LIN {X 0,Y 309.952,Z 757.671,A -85,B 0,C 180,E1 16400.5,E2 16400.5} C_VEL
LIN {X 0,Y 315.496,Z 768.364,A -85,B 0,C 180,E1 16405.207,E2 16405.207} C_VEL
LIN {X 0,Y 323.585,Z 785.947,A -85,B 0,C 180,E1 16410.491,E2 16410.491} C_VEL
LIN {X 0,Y 330.454,Z 808.188,A -85,B 0,C 180,E1 16415.117,E2 16415.117} C_VEL
LIN {X 0,Y 332.318,Z 818.689,A -85,B 0,C 180,E1 16416.877,E2 16416.877} C_VEL
LIN {X 0,Y 321.073,Z 855.454,A -85,B 0,C 180,E1 16419.899,E2 16419.899} C_VEL
LIN {X 0,Y 307.71,Z 890.699,A -85,B 0,C 180,E1 16424.174,E2 16424.174} C_VEL
LIN {X 0,Y 294.928,Z 920.705,A -85,B 0,C 180,E1 16429.49,E2 16429.49} C_VEL
LIN {X 0,Y 283.712,Z 946.43,A -85,B 0,C 180,E1 16435.988,E2 16435.988} C_VEL
LIN {X 0,Y 275.518,Z 966.441,A -85,B 0,C 180,E1 16443.137,E2 16443.137} C_VEL
LIN {X 0,Y 270.884,Z 980.87,A -85,B 0,C 180,E1 16450.473,E2 16450.473} C_VEL
LIN {X 0,Y 268.893,Z 991.255,A -85,B 0,C 180,E1 16458.671,E2 16458.671} C_VEL
LIN {X 0,Y 268.674,Z 996.154,A -85,B 0,C 180,E1 16466.78,E2 16466.78} C_VEL
LIN {X 0,Y 269.019,Z 996.603,A -85,B 0,C 180,E1 16470,E2 16470} C_VEL
LIN {X 0,Y 268.663,Z 993.875,A -85,B 0,C 180,E1 16478.072,E2 16478.072} C_VEL
LIN {X 0,Y 269.779,Z 985.621,A -85,B 0,C 180,E1 16486.241,E2 16486.241} C_VEL
LIN {X 0,Y 273.628,Z 971.419,A -85,B 0,C 180,E1 16494.444,E2 16494.444} C_VEL
LIN {X 0,Y 280.981,Z 951.52,A -85,B 0,C 180,E1 16502.08,E2 16502.08} C_VEL
LIN {X 0,Y 291.2,Z 926.496,A -85,B 0,C 180,E1 16508.747,E2 16508.747} C_VEL
LIN {X 0,Y 302.201,Z 899.005,A -85,B 0,C 180,E1 16513.938,E2 16513.938} C_VEL
LIN {X 0,Y 313.934,Z 866.938,A -85,B 0,C 180,E1 16518.208,E2 16518.208} C_VEL
LIN {X 0,Y 324.235,Z 833.113,A -85,B 0,C 180,E1 16521.361,E2 16521.361} C_VEL
LIN {X 0,Y 328.214,Z 816.116,A -85,B 0,C 180,E1 16522.625,E2 16522.625} C_VEL
LIN {X 0,Y 317.617,Z 786.468,A -85,B 0,C 180,E1 16527.572,E2 16527.572} C_VEL
LIN {X 0,Y 309.539,Z 769.18,A -85,B 0,C 180,E1 16530.843,E2 16530.843} C_VEL
LIN {X 0,Y 305.434,Z 765.763,A -85,B 0,C 180,E1 16532.16,E2 16532.16} C_VEL
LIN {X 0,Y 298.724,Z 762.182,A -85,B 0,C 180,E1 16534.27,E2 16534.27} C_VEL
LIN {X 0,Y 298.214,Z 761.313,A -85,B 0,C 180,E1 16534.479,E2 16534.479} C_VEL
LIN {X 0,Y 284.887,Z 739.622,A -85,B 0,C 180,E1 16540.243,E2 16540.243} C_VEL
LIN {X 0,Y 273.531,Z 723.276,A -85,B 0,C 180,E1 16545.909,E2 16545.909} C_VEL
LIN {X 0,Y 268.525,Z 716.432,A -85,B 0,C 180,E1 16548.856,E2 16548.856} C_VEL
LIN {X 0,Y 265.071,Z 710.925,A -85,B 0,C 180,E1 16551.193,E2 16551.193} C_VEL
LIN {X 0,Y 260.012,Z 704.969,A -85,B 0,C 180,E1 16554.98,E2 16554.98} C_VEL
LIN {X 0,Y 259.721,Z 702.53,A -85,B 0,C 180,E1 16555.809,E2 16555.809} C_VEL
LIN {X 0,Y 260.153,Z 702.53,A -85,B 0,C 180,E1 16559.973,E2 16559.973} C_VEL
LIN {X 0,Y 259.354,Z 702.53,A -85,B 0,C 180,E1 16568.46,E2 16568.46} C_VEL
LIN {X 0,Y 258.71,Z 702.53,A -85,B 0,C 180,E1 16576.924,E2 16576.924} C_VEL
LIN {X 0,Y 258.198,Z 702.53,A -85,B 0,C 180,E1 16584.113,E2 16584.113} C_VEL
LIN {X 0,Y 257.794,Z 702.53,A -85,B 0,C 180,E1 16591.751,E2 16591.751} C_VEL
LIN {X 0,Y 257.771,Z 703.057,A -85,B 0,C 180,E1 16597.239,E2 16597.239} C_VEL
LIN {X 0,Y 259.94,Z 708.124,A -85,B 0,C 180,E1 16599.361,E2 16599.361} C_VEL
LIN {X 0,Y 263.477,Z 711.105,A -85,B 0,C 180,E1 16601.928,E2 16601.928} C_VEL
LIN {X 0,Y 267.434,Z 716.658,A -85,B 0,C 180,E1 16604.625,E2 16604.625} C_VEL
LIN {X 0,Y 278.791,Z 731.981,A -85,B 0,C 180,E1 16611.013,E2 16611.013} C_VEL
LIN {X 0,Y 290.731,Z 751.396,A -85,B 0,C 180,E1 16617.012,E2 16617.012} C_VEL
LIN {X 0,Y 301.764,Z 773.502,A -85,B 0,C 180,E1 16622.492,E2 16622.492} C_VEL
LIN {X 0,Y 310.582,Z 798.842,A -85,B 0,C 180,E1 16627.717,E2 16627.717} C_VEL
LIN {X 0,Y 313.35,Z 812.889,A -85,B 0,C 180,E1 16630.3,E2 16630.3} C_VEL
LIN {X 0,Y 302.475,Z 846.573,A -85,B 0,C 180,E1 16634.075,E2 16634.075} C_VEL
LIN {X 0,Y 291.256,Z 875.538,A -85,B 0,C 180,E1 16638.797,E2 16638.797} C_VEL
LIN {X 0,Y 280.621,Z 900.044,A -85,B 0,C 180,E1 16644.533,E2 16644.533} C_VEL
LIN {X 0,Y 271.528,Z 920.415,A -85,B 0,C 180,E1 16651.468,E2 16651.468} C_VEL
LIN {X 0,Y 265.354,Z 935.057,A -85,B 0,C 180,E1 16658.959,E2 16658.959} C_VEL
LIN {X 0,Y 262.16,Z 944.332,A -85,B 0,C 180,E1 16666.727,E2 16666.727} C_VEL
LIN {X 0,Y 260.433,Z 948.523,A -85,B 0,C 180,E1 16673.929,E2 16673.929} C_VEL
LIN {X 0,Y 260.646,Z 948.698,A -85,B 0,C 180,E1 16681.404,E2 16681.404} C_VEL
LIN {X 0,Y 263.067,Z 944.4,A -85,B 0,C 180,E1 16689.124,E2 16689.124} C_VEL
LIN {X 0,Y 267.8,Z 934.327,A -85,B 0,C 180,E1 16697.501,E2 16697.501} C_VEL
LIN {X 0,Y 275.753,Z 918.84,A -85,B 0,C 180,E1 16705.171,E2 16705.171} C_VEL
LIN {X 0,Y 286.314,Z 898.705,A -85,B 0,C 180,E1 16711.718,E2 16711.718} C_VEL
LIN {X 0,Y 298.719,Z 873.349,A -85,B 0,C 180,E1 16717.371,E2 16717.371} C_VEL
LIN {X 0,Y 311.444,Z 844.042,A -85,B 0,C 180,E1 16721.852,E2 16721.852} C_VEL
LIN {X 0,Y 320.875,Z 817.036,A -85,B 0,C 180,E1 16724.861,E2 16724.861} C_VEL
LIN {X 0,Y 317.416,Z 795.177,A -85,B 0,C 180,E1 16729.755,E2 16729.755} C_VEL
LIN {X 0,Y 312.367,Z 777.587,A -85,B 0,C 180,E1 16734.827,E2 16734.827} C_VEL
LIN {X 0,Y 307.316,Z 764.973,A -85,B 0,C 180,E1 16740.239,E2 16740.239} C_VEL
LIN {X 0,Y 305.699,Z 761.257,A -85,B 0,C 180,E1 16742.579,E2 16742.579} C_VEL
LIN {X 0,Y 304.113,Z 756.55,A -85,B 0,C 180,E1 16746.2,E2 16746.2} C_VEL
LIN {X 0,Y 304.093,Z 757.322,A -85,B 0,C 180,E1 16754.463,E2 16754.463} C_VEL
LIN {X 0,Y 307.631,Z 765.127,A -85,B 0,C 180,E1 16760.204,E2 16760.204} C_VEL
LIN {X 0,Y 312.812,Z 776.006,A -85,B 0,C 180,E1 16765.025,E2 16765.025} C_VEL
LIN {X 0,Y 319.966,Z 793.22,A -85,B 0,C 180,E1 16770.23,E2 16770.23} C_VEL
LIN {X 0,Y 325.982,Z 815.534,A -85,B 0,C 180,E1 16774.947,E2 16774.947} C_VEL
LIN {X 0,Y 326.56,Z 822.504,A -85,B 0,C 180,E1 16776.018,E2 16776.018} C_VEL
LIN {X 0,Y 314.643,Z 858.935,A -85,B 0,C 180,E1 16779.172,E2 16779.172} C_VEL
LIN {X 0,Y 301.149,Z 892.374,A -85,B 0,C 180,E1 16783.399,E2 16783.399} C_VEL
LIN {X 0,Y 287.801,Z 922.182,A -85,B 0,C 180,E1 16788.882,E2 16788.882} C_VEL
LIN {X 0,Y 276.655,Z 946.385,A -85,B 0,C 180,E1 16795.212,E2 16795.212} C_VEL
LIN {X 0,Y 267.479,Z 967.633,A -85,B 0,C 180,E1 16803.17,E2 16803.17} C_VEL
LIN {X 0,Y 262.701,Z 981.909,A -85,B 0,C 180,E1 16811.046,E2 16811.046} C_VEL
LIN {X 0,Y 261.036,Z 990.52,A -85,B 0,C 180,E1 16818.282,E2 16818.282} C_VEL
LIN {X 0,Y 260.73,Z 994.111,A -85,B 0,C 180,E1 16823.352,E2 16823.352} C_VEL
LIN {X 0,Y 261.163,Z 995.89,A -85,B 0,C 180,E1 16830,E2 16830} C_VEL
LIN {X 0,Y 260.794,Z 993.127,A -85,B 0,C 180,E1 16838.317,E2 16838.317} C_VEL
LIN {X 0,Y 262.019,Z 984.826,A -85,B 0,C 180,E1 16846.735,E2 16846.735} C_VEL
LIN {X 0,Y 266.059,Z 970.858,A -85,B 0,C 180,E1 16855.021,E2 16855.021} C_VEL
LIN {X 0,Y 273.951,Z 950.669,A -85,B 0,C 180,E1 16862.953,E2 16862.953} C_VEL
LIN {X 0,Y 284.345,Z 926.389,A -85,B 0,C 180,E1 16869.556,E2 16869.556} C_VEL
LIN {X 0,Y 296.508,Z 897.188,A -85,B 0,C 180,E1 16875.123,E2 16875.123} C_VEL
LIN {X 0,Y 308.405,Z 865.604,A -85,B 0,C 180,E1 16879.324,E2 16879.324} C_VEL
LIN {X 0,Y 319.029,Z 831.642,A -85,B 0,C 180,E1 16882.465,E2 16882.465} C_VEL
LIN {X 0,Y 322.022,Z 818.898,A -85,B 0,C 180,E1 16883.439,E2 16883.439} C_VEL
LIN {X 0,Y 312.462,Z 791.073,A -85,B 0,C 180,E1 16888.3,E2 16888.3} C_VEL
LIN {X 0,Y 299.497,Z 763.712,A -85,B 0,C 180,E1 16893.922,E2 16893.922} C_VEL
LIN {X 0,Y 298.214,Z 761.313,A -85,B 0,C 180,E1 16894.479,E2 16894.479} C_VEL
LIN {X 0,Y 292.885,Z 755.46,A -85,B 0,C 180,E1 16896.496,E2 16896.496} C_VEL
LIN {X 0,Y 283.364,Z 748.358,A -85,B 0,C 180,E1 16900.231,E2 16900.231} C_VEL
LIN {X 0,Y 271.288,Z 730.388,A -85,B 0,C 180,E1 16906.474,E2 16906.474} C_VEL
LIN {X 0,Y 265.81,Z 723.086,A -85,B 0,C 180,E1 16909.8,E2 16909.8} C_VEL
LIN {X 0,Y 261.859,Z 717.005,A -85,B 0,C 180,E1 16912.634,E2 16912.634} C_VEL
LIN {X 0,Y 257.895,Z 711.36,A -85,B 0,C 180,E1 16915.885,E2 16915.885} C_VEL
LIN {X 0,Y 255.967,Z 709.404,A -85,B 0,C 180,E1 16917.586,E2 16917.586} C_VEL
LIN {X 0,Y 252.121,Z 703.78,A -85,B 0,C 180,E1 16921.901,E2 16921.901} C_VEL
LIN {X 0,Y 252.032,Z 702.53,A -85,B 0,C 180,E1 16922.546,E2 16922.546} C_VEL
LIN {X 0,Y 251.304,Z 702.53,A -85,B 0,C 180,E1 16930.348,E2 16930.348} C_VEL
LIN {X 0,Y 250.706,Z 702.53,A -85,B 0,C 180,E1 16937.482,E2 16937.482} C_VEL
LIN {X 0,Y 250.123,Z 702.53,A -85,B 0,C 180,E1 16945.182,E2 16945.182} C_VEL
LIN {X 0,Y 249.917,Z 703.282,A -85,B 0,C 180,E1 16949.517,E2 16949.517} C_VEL
LIN {X 0,Y 252.514,Z 708.484,A -85,B 0,C 180,E1 16953.302,E2 16953.302} C_VEL
LIN {X 0,Y 255.955,Z 711.064,A -85,B 0,C 180,E1 16956.691,E2 16956.691} C_VEL
LIN {X 0,Y 259.601,Z 716.781,A -85,B 0,C 180,E1 16959.968,E2 16959.968} C_VEL
LIN {X 0,Y 261.694,Z 719.033,A -85,B 0,C 180,E1 16961.535,E2 16961.535} C_VEL
LIN {X 0,Y 267.398,Z 727.187,A -85,B 0,C 180,E1 16965.485,E2 16965.485} C_VEL
LIN {X 0,Y 276.033,Z 739.146,A -85,B 0,C 180,E1 16970.543,E2 16970.543} C_VEL
LIN {X 0,Y 287.79,Z 759.139,A -85,B 0,C 180,E1 16976.872,E2 16976.872} C_VEL
LIN {X 0,Y 297.989,Z 781.572,A -85,B 0,C 180,E1 16982.479,E2 16982.479} C_VEL
LIN {X 0,Y 305.562,Z 805.841,A -85,B 0,C 180,E1 16987.618,E2 16987.618} C_VEL
LIN {X 0,Y 307.052,Z 816.176,A -85,B 0,C 180,E1 16989.514,E2 16989.514} C_VEL
LIN {X 0,Y 295.398,Z 850.222,A -85,B 0,C 180,E1 16993.492,E2 16993.492} C_VEL
LIN {X 0,Y 283.523,Z 879.262,A -85,B 0,C 180,E1 16998.487,E2 16998.487} C_VEL
LIN {X 0,Y 272.351,Z 904.007,A -85,B 0,C 180,E1 17004.666,E2 17004.666} C_VEL
LIN {X 0,Y 263.492,Z 922.835,A -85,B 0,C 180,E1 17011.512,E2 17011.512} C_VEL
LIN {X 0,Y 257.221,Z 937.08,A -85,B 0,C 180,E1 17019.392,E2 17019.392} C_VEL
LIN {X 0,Y 254.111,Z 945.653,A -85,B 0,C 180,E1 17027.273,E2 17027.273} C_VEL
LIN {X 0,Y 252.449,Z 949.511,A -85,B 0,C 180,E1 17034.736,E2 17034.736} C_VEL
LIN {X 0,Y 253.221,Z 948.827,A -85,B 0,C 180,E1 17043.527,E2 17043.527} C_VEL
LIN {X 0,Y 255.721,Z 944.406,A -85,B 0,C 180,E1 17050.476,E2 17050.476} C_VEL
LIN {X 0,Y 260.915,Z 934.25,A -85,B 0,C 180,E1 17058.753,E2 17058.753} C_VEL
LIN {X 0,Y 269.311,Z 919,A -85,B 0,C 180,E1 17066.295,E2 17066.295} C_VEL
LIN {X 0,Y 280.66,Z 898.461,A -85,B 0,C 180,E1 17073.015,E2 17073.015} C_VEL
LIN {X 0,Y 293.25,Z 873.912,A -85,B 0,C 180,E1 17078.513,E2 17078.513} C_VEL
LIN {X 0,Y 306.964,Z 843.551,A -85,B 0,C 180,E1 17083.153,E2 17083.153} C_VEL
LIN {X 0,Y 315.393,Z 819.76,A -85,B 0,C 180,E1 17085.892,E2 17085.892} C_VEL
LIN {X 0,Y 312.425,Z 798.271,A -85,B 0,C 180,E1 17090.993,E2 17090.993} C_VEL
LIN {X 0,Y 308.013,Z 781.769,A -85,B 0,C 180,E1 17096.224,E2 17096.224} C_VEL
LIN {X 0,Y 303.922,Z 769.5,A -85,B 0,C 180,E1 17101.908,E2 17101.908} C_VEL
LIN {X 0,Y 301.889,Z 764.119,A -85,B 0,C 180,E1 17106.733,E2 17106.733} C_VEL
LIN {X 0,Y 302.054,Z 764.998,A -85,B 0,C 180,E1 17114.258,E2 17114.258} C_VEL
LIN {X 0,Y 305.197,Z 772.567,A -85,B 0,C 180,E1 17119.964,E2 17119.964} C_VEL
LIN {X 0,Y 310.416,Z 784.431,A -85,B 0,C 180,E1 17125.192,E2 17125.192} C_VEL
LIN {X 0,Y 316.779,Z 802.18,A -85,B 0,C 180,E1 17130.426,E2 17130.426} C_VEL
LIN {X 0,Y 321.468,Z 823.556,A -85,B 0,C 180,E1 17134.913,E2 17134.913} C_VEL
LIN {X 0,Y 308.737,Z 860.849,A -85,B 0,C 180,E1 17138.245,E2 17138.245} C_VEL
LIN {X 0,Y 295.1,Z 893.08,A -85,B 0,C 180,E1 17142.425,E2 17142.425} C_VEL
LIN {X 0,Y 281.395,Z 922.208,A -85,B 0,C 180,E1 17147.907,E2 17147.907} C_VEL
LIN {X 0,Y 269.669,Z 946.291,A -85,B 0,C 180,E1 17154.376,E2 17154.376} C_VEL
LIN {X 0,Y 260.182,Z 966.977,A -85,B 0,C 180,E1 17162.355,E2 17162.355} C_VEL
LIN {X 0,Y 254.987,Z 981.316,A -85,B 0,C 180,E1 17170.512,E2 17170.512} C_VEL
LIN {X 0,Y 253.174,Z 989.86,A -85,B 0,C 180,E1 17177.958,E2 17177.958} C_VEL
LIN {X 0,Y 252.865,Z 993.419,A -85,B 0,C 180,E1 17183.145,E2 17183.145} C_VEL
LIN {X 0,Y 253.293,Z 995.176,A -85,B 0,C 180,E1 17190,E2 17190} C_VEL
LIN {X 0,Y 252.915,Z 992.371,A -85,B 0,C 180,E1 17198.578,E2 17198.578} C_VEL
LIN {X 0,Y 254.261,Z 984.005,A -85,B 0,C 180,E1 17207.262,E2 17207.262} C_VEL
LIN {X 0,Y 258.795,Z 969.492,A -85,B 0,C 180,E1 17216.009,E2 17216.009} C_VEL
LIN {X 0,Y 267.032,Z 949.646,A -85,B 0,C 180,E1 17223.92,E2 17223.92} C_VEL
LIN {X 0,Y 278.05,Z 925.23,A -85,B 0,C 180,E1 17230.636,E2 17230.636} C_VEL
LIN {X 0,Y 290.412,Z 896.619,A -85,B 0,C 180,E1 17236.149,E2 17236.149} C_VEL
LIN {X 0,Y 302.589,Z 865.36,A -85,B 0,C 180,E1 17240.342,E2 17240.342} C_VEL
LIN {X 0,Y 314.007,Z 829.906,A -85,B 0,C 180,E1 17243.622,E2 17243.622} C_VEL
LIN {X 0,Y 315.829,Z 821.525,A -85,B 0,C 180,E1 17244.316,E2 17244.316} C_VEL
LIN {X 0,Y 306.732,Z 794.337,A -85,B 0,C 180,E1 17249.29,E2 17249.29} C_VEL
LIN {X 0,Y 294.241,Z 767.159,A -85,B 0,C 180,E1 17255.152,E2 17255.152} C_VEL
LIN {X 0,Y 283.364,Z 748.358,A -85,B 0,C 180,E1 17260.231,E2 17260.231} C_VEL
LIN {X 0,Y 276.578,Z 742.524,A -85,B 0,C 180,E1 17263.301,E2 17263.301} C_VEL
LIN {X 0,Y 269.757,Z 738.248,A -85,B 0,C 180,E1 17266.613,E2 17266.613} C_VEL
LIN {X 0,Y 259.79,Z 724.228,A -85,B 0,C 180,E1 17273.303,E2 17273.303} C_VEL
LIN {X 0,Y 255.908,Z 718.162,A -85,B 0,C 180,E1 17276.669,E2 17276.669} C_VEL
LIN {X 0,Y 250.725,Z 711.765,A -85,B 0,C 180,E1 17282.235,E2 17282.235} C_VEL
LIN {X 0,Y 249.92,Z 710.151,A -85,B 0,C 180,E1 17283.433,E2 17283.433} C_VEL
LIN {X 0,Y 244.951,Z 707.669,A -85,B 0,C 180,E1 17294.233,E2 17294.233} C_VEL
LIN {X 0,Y 248.352,Z 710.423,A -85,B 0,C 180,E1 17308.742,E2 17308.742} C_VEL
LIN {X 0,Y 251.252,Z 716.251,A -85,B 0,C 180,E1 17313.123,E2 17313.123} C_VEL
LIN {X 0,Y 254.28,Z 718.794,A -85,B 0,C 180,E1 17316.226,E2 17316.226} C_VEL
LIN {X 0,Y 258.378,Z 724.622,A -85,B 0,C 180,E1 17319.928,E2 17319.928} C_VEL
LIN {X 0,Y 265.434,Z 734.864,A -85,B 0,C 180,E1 17325.172,E2 17325.172} C_VEL
LIN {X 0,Y 273.871,Z 747.567,A -85,B 0,C 180,E1 17330.502,E2 17330.502} C_VEL
LIN {X 0,Y 283.765,Z 765.176,A -85,B 0,C 180,E1 17336.237,E2 17336.237} C_VEL
LIN {X 0,Y 292.976,Z 786.556,A -85,B 0,C 180,E1 17341.778,E2 17341.778} C_VEL
LIN {X 0,Y 299.743,Z 809.701,A -85,B 0,C 180,E1 17346.885,E2 17346.885} C_VEL
LIN {X 0,Y 300.903,Z 819.016,A -85,B 0,C 180,E1 17348.658,E2 17348.658} C_VEL
LIN {X 0,Y 288.794,Z 852.607,A -85,B 0,C 180,E1 17352.712,E2 17352.712} C_VEL
LIN {X 0,Y 276.601,Z 881.237,A -85,B 0,C 180,E1 17357.796,E2 17357.796} C_VEL
LIN {X 0,Y 264.9,Z 906.018,A -85,B 0,C 180,E1 17364.221,E2 17364.221} C_VEL
LIN {X 0,Y 255.917,Z 924.145,A -85,B 0,C 180,E1 17371.114,E2 17371.114} C_VEL
LIN {X 0,Y 249.212,Z 938.66,A -85,B 0,C 180,E1 17379.586,E2 17379.586} C_VEL
LIN {X 0,Y 246.057,Z 946.935,A -85,B 0,C 180,E1 17387.857,E2 17387.857} C_VEL
LIN {X 0,Y 244.507,Z 950.35,A -85,B 0,C 180,E1 17395.596,E2 17395.596} C_VEL
LIN {X 0,Y 245.381,Z 949.643,A -85,B 0,C 180,E1 17403.606,E2 17403.606} C_VEL
LIN {X 0,Y 248.46,Z 944.323,A -85,B 0,C 180,E1 17411.92,E2 17411.92} C_VEL
LIN {X 0,Y 254.508,Z 933.497,A -85,B 0,C 180,E1 17420.426,E2 17420.426} C_VEL
LIN {X 0,Y 263.868,Z 917.609,A -85,B 0,C 180,E1 17428.111,E2 17428.111} C_VEL
LIN {X 0,Y 276.714,Z 895.521,A -85,B 0,C 180,E1 17435.106,E2 17435.106} C_VEL
LIN {X 0,Y 290.617,Z 869.15,A -85,B 0,C 180,E1 17440.664,E2 17440.664} C_VEL
LIN {X 0,Y 304.031,Z 839.579,A -85,B 0,C 180,E1 17444.915,E2 17444.915} C_VEL
LIN {X 0,Y 310.084,Z 823.602,A -85,B 0,C 180,E1 17446.732,E2 17446.732} C_VEL
LIN {X 0,Y 307.824,Z 802.789,A -85,B 0,C 180,E1 17451.923,E2 17451.923} C_VEL
LIN {X 0,Y 304.146,Z 787.118,A -85,B 0,C 180,E1 17457.18,E2 17457.18} C_VEL
LIN {X 0,Y 300.784,Z 776.165,A -85,B 0,C 180,E1 17462.898,E2 17462.898} C_VEL
LIN {X 0,Y 299.708,Z 771.704,A -85,B 0,C 180,E1 17466.527,E2 17466.527} C_VEL
LIN {X 0,Y 299.751,Z 772.559,A -85,B 0,C 180,E1 17474.071,E2 17474.071} C_VEL
LIN {X 0,Y 302.518,Z 779.708,A -85,B 0,C 180,E1 17479.581,E2 17479.581} C_VEL
LIN {X 0,Y 307.375,Z 792.005,A -85,B 0,C 180,E1 17485.07,E2 17485.07} C_VEL
LIN {X 0,Y 312.916,Z 809.903,A -85,B 0,C 180,E1 17490.307,E2 17490.307} C_VEL
LIN {X 0,Y 315.904,Z 826.108,A -85,B 0,C 180,E1 17493.842,E2 17493.842} C_VEL
LIN {X 0,Y 303.741,Z 860.867,A -85,B 0,C 180,E1 17497.084,E2 17497.084} C_VEL
LIN {X 0,Y 289.793,Z 892.456,A -85,B 0,C 180,E1 17501.198,E2 17501.198} C_VEL
LIN {X 0,Y 275.329,Z 921.716,A -85,B 0,C 180,E1 17506.756,E2 17506.756} C_VEL
LIN {X 0,Y 262.621,Z 946.496,A -85,B 0,C 180,E1 17513.582,E2 17513.582} C_VEL
LIN {X 0,Y 252.957,Z 966.354,A -85,B 0,C 180,E1 17521.494,E2 17521.494} C_VEL
LIN {X 0,Y 246.907,Z 982.098,A -85,B 0,C 180,E1 17530.925,E2 17530.925} C_VEL
LIN {X 0,Y 245.083,Z 991.181,A -85,B 0,C 180,E1 17540.201,E2 17540.201} C_VEL
LIN {X 0,Y 245,Z 994.042,A -85,B 0,C 180,E1 17546.468,E2 17546.468} C_VEL
LIN {X 0,Y 245.435,Z 994.461,A -85,B 0,C 180,E1 17550,E2 17550} C_VEL
LIN {X 0,Y 244.987,Z 992.571,A -85,B 0,C 180,E1 17557.076,E2 17557.076} C_VEL
LIN {X 0,Y 245.63,Z 987.23,A -85,B 0,C 180,E1 17564.225,E2 17564.225} C_VEL
LIN {X 0,Y 248.901,Z 975.286,A -85,B 0,C 180,E1 17573.208,E2 17573.208} C_VEL
LIN {X 0,Y 256.434,Z 956.837,A -85,B 0,C 180,E1 17581.979,E2 17581.979} C_VEL
LIN {X 0,Y 267.09,Z 933.964,A -85,B 0,C 180,E1 17589.322,E2 17589.322} C_VEL
LIN {X 0,Y 279.965,Z 906.038,A -85,B 0,C 180,E1 17595.495,E2 17595.495} C_VEL
LIN {X 0,Y 292.999,Z 875.279,A -85,B 0,C 180,E1 17600.182,E2 17600.182} C_VEL
LIN {X 0,Y 304.946,Z 841.582,A -85,B 0,C 180,E1 17603.747,E2 17603.747} C_VEL
LIN {X 0,Y 309.885,Z 824.82,A -85,B 0,C 180,E1 17605.101,E2 17605.101} C_VEL
LIN {X 0,Y 301.092,Z 797.494,A -85,B 0,C 180,E1 17610.317,E2 17610.317} C_VEL
LIN {X 0,Y 288.674,Z 769.981,A -85,B 0,C 180,E1 17616.592,E2 17616.592} C_VEL
LIN {X 0,Y 275.983,Z 748.133,A -85,B 0,C 180,E1 17623.091,E2 17623.091} C_VEL
LIN {X 0,Y 269.757,Z 738.248,A -85,B 0,C 180,E1 17626.613,E2 17626.613} C_VEL
LIN {X 0,Y 258.21,Z 731.808,A -85,B 0,C 180,E1 17633.643,E2 17633.643} C_VEL
LIN {X 0,Y 253.05,Z 724.683,A -85,B 0,C 180,E1 17638.264,E2 17638.264} C_VEL
LIN {X 0,Y 248.84,Z 717.96,A -85,B 0,C 180,E1 17643.448,E2 17643.448} C_VEL
LIN {X 0,Y 243.879,Z 715.499,A -85,B 0,C 180,E1 17654.297,E2 17654.297} C_VEL
LIN {X 0,Y 246.955,Z 718.182,A -85,B 0,C 180,E1 17668.28,E2 17668.28} C_VEL
LIN {X 0,Y 250.535,Z 724.433,A -85,B 0,C 180,E1 17673.557,E2 17673.557} C_VEL
LIN {X 0,Y 252.651,Z 726.565,A -85,B 0,C 180,E1 17675.835,E2 17675.835} C_VEL
LIN {X 0,Y 258.317,Z 734.997,A -85,B 0,C 180,E1 17681.04,E2 17681.04} C_VEL
LIN {X 0,Y 266.292,Z 746.827,A -85,B 0,C 180,E1 17686.978,E2 17686.978} C_VEL
LIN {X 0,Y 276.421,Z 764.625,A -85,B 0,C 180,E1 17693.581,E2 17693.581} C_VEL
LIN {X 0,Y 285.997,Z 785.88,A -85,B 0,C 180,E1 17699.704,E2 17699.704} C_VEL
LIN {X 0,Y 293.135,Z 809.737,A -85,B 0,C 180,E1 17705.315,E2 17705.315} C_VEL
LIN {X 0,Y 294.696,Z 821.987,A -85,B 0,C 180,E1 17707.799,E2 17707.799} C_VEL
LIN {X 0,Y 282.752,Z 853.793,A -85,B 0,C 180,E1 17711.727,E2 17711.727} C_VEL
LIN {X 0,Y 270.433,Z 881.631,A -85,B 0,C 180,E1 17716.737,E2 17716.737} C_VEL
LIN {X 0,Y 258.102,Z 906.67,A -85,B 0,C 180,E1 17723.324,E2 17723.324} C_VEL
LIN {X 0,Y 248.302,Z 925.503,A -85,B 0,C 180,E1 17730.722,E2 17730.722} C_VEL
LIN {X 0,Y 241.656,Z 939.199,A -85,B 0,C 180,E1 17738.982,E2 17738.982} C_VEL
LIN {X 0,Y 238.602,Z 946.777,A -85,B 0,C 180,E1 17746.382,E2 17746.382} C_VEL
LIN {X 0,Y 236.947,Z 950.212,A -85,B 0,C 180,E1 17752.465,E2 17752.465} C_VEL
LIN {X 0,Y 236.854,Z 951.194,A -85,B 0,C 180,E1 17760.644,E2 17760.644} C_VEL
LIN {X 0,Y 239.432,Z 947.77,A -85,B 0,C 180,E1 17769.069,E2 17769.069} C_VEL
LIN {X 0,Y 244.935,Z 938.247,A -85,B 0,C 180,E1 17778.562,E2 17778.562} C_VEL
LIN {X 0,Y 253.443,Z 924.575,A -85,B 0,C 180,E1 17786.469,E2 17786.469} C_VEL
LIN {X 0,Y 265.227,Z 905.679,A -85,B 0,C 180,E1 17793.589,E2 17793.589} C_VEL
LIN {X 0,Y 279.832,Z 880.572,A -85,B 0,C 180,E1 17799.879,E2 17799.879} C_VEL
LIN {X 0,Y 294.79,Z 850.899,A -85,B 0,C 180,E1 17804.799,E2 17804.799} C_VEL
LIN {X 0,Y 304.568,Z 827.906,A -85,B 0,C 180,E1 17807.525,E2 17807.525} C_VEL
LIN {X 0,Y 303.517,Z 809.682,A -85,B 0,C 180,E1 17812.167,E2 17812.167} C_VEL
LIN {X 0,Y 300.914,Z 794.958,A -85,B 0,C 180,E1 17817.149,E2 17817.149} C_VEL
LIN {X 0,Y 298.117,Z 783.656,A -85,B 0,C 180,E1 17822.924,E2 17822.924} C_VEL
LIN {X 0,Y 297.227,Z 780.292,A -85,B 0,C 180,E1 17825.85,E2 17825.85} C_VEL
LIN {X 0,Y 296.852,Z 779.072,A -85,B 0,C 180,E1 17831.753,E2 17831.753} C_VEL
LIN {X 0,Y 297.389,Z 781.231,A -85,B 0,C 180,E1 17834.718,E2 17834.718} C_VEL
LIN {X 0,Y 299.554,Z 786.632,A -85,B 0,C 180,E1 17839.133,E2 17839.133} C_VEL
LIN {X 0,Y 303.771,Z 798.613,A -85,B 0,C 180,E1 17844.609,E2 17844.609} C_VEL
LIN {X 0,Y 308.305,Z 815.126,A -85,B 0,C 180,E1 17849.622,E2 17849.622} C_VEL
LIN {X 0,Y 310.551,Z 830.396,A -85,B 0,C 180,E1 17853.046,E2 17853.046} C_VEL
LIN {X 0,Y 296.032,Z 867.528,A -85,B 0,C 180,E1 17856.595,E2 17856.595} C_VEL
LIN {X 0,Y 280.858,Z 899.613,A -85,B 0,C 180,E1 17861.217,E2 17861.217} C_VEL
LIN {X 0,Y 266.023,Z 927.583,A -85,B 0,C 180,E1 17867.101,E2 17867.101} C_VEL
LIN {X 0,Y 253.057,Z 951.454,A -85,B 0,C 180,E1 17874.45,E2 17874.45} C_VEL
LIN {X 0,Y 244.102,Z 969.194,A -85,B 0,C 180,E1 17882.377,E2 17882.377} C_VEL
LIN {X 0,Y 238.762,Z 982.931,A -85,B 0,C 180,E1 17891.578,E2 17891.578} C_VEL
LIN {X 0,Y 237.185,Z 990.735,A -85,B 0,C 180,E1 17900.3,E2 17900.3} C_VEL
LIN {X 0,Y 237.119,Z 993.335,A -85,B 0,C 180,E1 17906.351,E2 17906.351} C_VEL
LIN {X 0,Y 237.554,Z 993.743,A -85,B 0,C 180,E1 17910,E2 17910} C_VEL
LIN {X 0,Y 237.096,Z 991.824,A -85,B 0,C 180,E1 17917.313,E2 17917.313} C_VEL
LIN {X 0,Y 237.817,Z 986.439,A -85,B 0,C 180,E1 17924.703,E2 17924.703} C_VEL
LIN {X 0,Y 241.404,Z 974.438,A -85,B 0,C 180,E1 17933.954,E2 17933.954} C_VEL
LIN {X 0,Y 249.488,Z 955.839,A -85,B 0,C 180,E1 17942.981,E2 17942.981} C_VEL
LIN {X 0,Y 260.417,Z 933.477,A -85,B 0,C 180,E1 17950.29,E2 17950.29} C_VEL
LIN {X 0,Y 273.358,Z 906.534,A -85,B 0,C 180,E1 17956.388,E2 17956.388} C_VEL
LIN {X 0,Y 286.856,Z 875.932,A -85,B 0,C 180,E1 17961.15,E2 17961.15} C_VEL
LIN {X 0,Y 299.118,Z 842.613,A -85,B 0,C 180,E1 17964.74,E2 17964.74} C_VEL
LIN {X 0,Y 303.634,Z 827.168,A -85,B 0,C 180,E1 17966.07,E2 17966.07} C_VEL
LIN {X 0,Y 295.394,Z 800.539,A -85,B 0,C 180,E1 17971.416,E2 17971.416} C_VEL
LIN {X 0,Y 283.439,Z 773.178,A -85,B 0,C 180,E1 17977.995,E2 17977.995} C_VEL
LIN {X 0,Y 270.793,Z 751.017,A -85,B 0,C 180,E1 17985.043,E2 17985.043} C_VEL
LIN {X 0,Y 261.633,Z 737.407,A -85,B 0,C 180,E1 17990.958,E2 17990.958} C_VEL
LIN {X 0,Y 258.21,Z 731.808,A -85,B 0,C 180,E1 17993.643,E2 17993.643} C_VEL
LIN {X 0,Y 251.442,Z 732.191,A -85,B 0,C 180,E1 17998.751,E2 17998.751} C_VEL
LIN {X 0,Y 247.06,Z 725.635,A -85,B 0,C 180,E1 18004.35,E2 18004.35} C_VEL
LIN {X 0,Y 242.806,Z 723.33,A -85,B 0,C 180,E1 18014.362,E2 18014.362} C_VEL
LIN {X 0,Y 245.622,Z 725.973,A -85,B 0,C 180,E1 18027.905,E2 18027.905} C_VEL
LIN {X 0,Y 249.21,Z 732.233,A -85,B 0,C 180,E1 18033.499,E2 18033.499} C_VEL
LIN {X 0,Y 251.062,Z 734.6,A -85,B 0,C 180,E1 18035.607,E2 18035.607} C_VEL
LIN {X 0,Y 256.154,Z 742.534,A -85,B 0,C 180,E1 18040.679,E2 18040.679} C_VEL
LIN {X 0,Y 263.61,Z 754.241,A -85,B 0,C 180,E1 18046.649,E2 18046.649} C_VEL
LIN {X 0,Y 272.77,Z 771.406,A -85,B 0,C 180,E1 18053.136,E2 18053.136} C_VEL
LIN {X 0,Y 281.241,Z 791.351,A -85,B 0,C 180,E1 18059.077,E2 18059.077} C_VEL
LIN {X 0,Y 287.667,Z 815.154,A -85,B 0,C 180,E1 18064.896,E2 18064.896} C_VEL
LIN {X 0,Y 288.708,Z 824.515,A -85,B 0,C 180,E1 18066.867,E2 18066.867} C_VEL
LIN {X 0,Y 276.297,Z 856.121,A -85,B 0,C 180,E1 18070.871,E2 18070.871} C_VEL
LIN {X 0,Y 263.01,Z 884.824,A -85,B 0,C 180,E1 18076.241,E2 18076.241} C_VEL
LIN {X 0,Y 250.237,Z 909.317,A -85,B 0,C 180,E1 18083.073,E2 18083.073} C_VEL
LIN {X 0,Y 240.106,Z 928.004,A -85,B 0,C 180,E1 18090.901,E2 18090.901} C_VEL
LIN {X 0,Y 233.586,Z 940.915,A -85,B 0,C 180,E1 18099.295,E2 18099.295} C_VEL
LIN {X 0,Y 230.547,Z 947.987,A -85,B 0,C 180,E1 18106.876,E2 18106.876} C_VEL
LIN {X 0,Y 228.911,Z 951.202,A -85,B 0,C 180,E1 18113.3,E2 18113.3} C_VEL
LIN {X 0,Y 229.15,Z 951.72,A -85,B 0,C 180,E1 18121.792,E2 18121.792} C_VEL
LIN {X 0,Y 232.117,Z 947.819,A -85,B 0,C 180,E1 18130.551,E2 18130.551} C_VEL
LIN {X 0,Y 237.858,Z 938.751,A -85,B 0,C 180,E1 18139.58,E2 18139.58} C_VEL
LIN {X 0,Y 248.062,Z 923.463,A -85,B 0,C 180,E1 18148.393,E2 18148.393} C_VEL
LIN {X 0,Y 261.649,Z 902.794,A -85,B 0,C 180,E1 18155.871,E2 18155.871} C_VEL
LIN {X 0,Y 276.918,Z 877.168,A -85,B 0,C 180,E1 18161.94,E2 18161.94} C_VEL
LIN {X 0,Y 292.286,Z 847.303,A -85,B 0,C 180,E1 18166.646,E2 18166.646} C_VEL
LIN {X 0,Y 299.529,Z 830.025,A -85,B 0,C 180,E1 18168.769,E2 18168.769} C_VEL
LIN {X 0,Y 298.658,Z 811.76,A -85,B 0,C 180,E1 18173.861,E2 18173.861} C_VEL
LIN {X 0,Y 296.434,Z 797.746,A -85,B 0,C 180,E1 18179.294,E2 18179.294} C_VEL
LIN {X 0,Y 294.672,Z 789.557,A -85,B 0,C 180,E1 18184.428,E2 18184.428} C_VEL
LIN {X 0,Y 294.116,Z 786.419,A -85,B 0,C 180,E1 18188.876,E2 18188.876} C_VEL
LIN {X 0,Y 294.544,Z 787.121,A -85,B 0,C 180,E1 18193.238,E2 18193.238} C_VEL
LIN {X 0,Y 296.463,Z 793.323,A -85,B 0,C 180,E1 18198.57,E2 18198.57} C_VEL
LIN {X 0,Y 300.15,Z 805.376,A -85,B 0,C 180,E1 18204.218,E2 18204.218} C_VEL
LIN {X 0,Y 303.928,Z 821.878,A -85,B 0,C 180,E1 18209.313,E2 18209.313} C_VEL
LIN {X 0,Y 305.018,Z 834.215,A -85,B 0,C 180,E1 18212.087,E2 18212.087} C_VEL
LIN {X 0,Y 290.133,Z 869.93,A -85,B 0,C 180,E1 18215.641,E2 18215.641} C_VEL
LIN {X 0,Y 275.55,Z 899.29,A -85,B 0,C 180,E1 18219.941,E2 18219.941} C_VEL
LIN {X 0,Y 260.08,Z 927.128,A -85,B 0,C 180,E1 18225.872,E2 18225.872} C_VEL
LIN {X 0,Y 246.406,Z 950.901,A -85,B 0,C 180,E1 18233.337,E2 18233.337} C_VEL
LIN {X 0,Y 236.857,Z 968.579,A -85,B 0,C 180,E1 18241.456,E2 18241.456} C_VEL
LIN {X 0,Y 231.088,Z 982.275,A -85,B 0,C 180,E1 18250.943,E2 18250.943} C_VEL
LIN {X 0,Y 229.421,Z 989.178,A -85,B 0,C 180,E1 18258.619,E2 18258.619} C_VEL
LIN {X 0,Y 229.224,Z 992.625,A -85,B 0,C 180,E1 18266.225,E2 18266.225} C_VEL
LIN {X 0,Y 229.694,Z 993.027,A -85,B 0,C 180,E1 18270,E2 18270} C_VEL
LIN {X 0,Y 229.243,Z 990.376,A -85,B 0,C 180,E1 18278.999,E2 18278.999} C_VEL
LIN {X 0,Y 230.827,Z 982.648,A -85,B 0,C 180,E1 18288.061,E2 18288.061} C_VEL
LIN {X 0,Y 236.036,Z 968.655,A -85,B 0,C 180,E1 18297.613,E2 18297.613} C_VEL
LIN {X 0,Y 245.512,Z 949.036,A -85,B 0,C 180,E1 18306.248,E2 18306.248} C_VEL
LIN {X 0,Y 258.237,Z 924.411,A -85,B 0,C 180,E1 18313.536,E2 18313.536} C_VEL
LIN {X 0,Y 272.237,Z 895.608,A -85,B 0,C 180,E1 18319.35,E2 18319.35} C_VEL
LIN {X 0,Y 286.388,Z 862.622,A -85,B 0,C 180,E1 18323.864,E2 18323.864} C_VEL
LIN {X 0,Y 297.583,Z 830.187,A -85,B 0,C 180,E1 18326.944,E2 18326.944} C_VEL
LIN {X 0,Y 289.761,Z 803.982,A -85,B 0,C 180,E1 18332.451,E2 18332.451} C_VEL
LIN {X 0,Y 278.846,Z 778.144,A -85,B 0,C 180,E1 18338.975,E2 18338.975} C_VEL
LIN {X 0,Y 267.578,Z 757.348,A -85,B 0,C 180,E1 18345.86,E2 18345.86} C_VEL
LIN {X 0,Y 258.447,Z 742.987,A -85,B 0,C 180,E1 18352.33,E2 18352.33} C_VEL
LIN {X 0,Y 255.241,Z 738.136,A -85,B 0,C 180,E1 18354.992,E2 18354.992} C_VEL
LIN {X 0,Y 251.442,Z 732.191,A -85,B 0,C 180,E1 18358.751,E2 18358.751} C_VEL
LIN {X 0,Y 247.587,Z 731.812,A -85,B 0,C 180,E1 18362.705,E2 18362.705} C_VEL
LIN {X 0,Y 244.357,Z 732.794,A -85,B 0,C 180,E1 18366.787,E2 18366.787} C_VEL
LIN {X 0,Y 241.445,Z 731.302,A -85,B 0,C 180,E1 18378.175,E2 18378.175} C_VEL
LIN {X 0,Y 244.294,Z 734.348,A -85,B 0,C 180,E1 18387.934,E2 18387.934} C_VEL
LIN {X 0,Y 248.2,Z 740.318,A -85,B 0,C 180,E1 18393.993,E2 18393.993} C_VEL
LIN {X 0,Y 254.104,Z 750.401,A -85,B 0,C 180,E1 18400.551,E2 18400.551} C_VEL
LIN {X 0,Y 261.549,Z 763.045,A -85,B 0,C 180,E1 18406.951,E2 18406.951} C_VEL
LIN {X 0,Y 270.544,Z 781.416,A -85,B 0,C 180,E1 18413.826,E2 18413.826} C_VEL
LIN {X 0,Y 277.634,Z 800.922,A -85,B 0,C 180,E1 18419.544,E2 18419.544} C_VEL
LIN {X 0,Y 282.594,Z 823.32,A -85,B 0,C 180,E1 18425.113,E2 18425.113} C_VEL
LIN {X 0,Y 282.218,Z 828.475,A -85,B 0,C 180,E1 18426.043,E2 18426.043} C_VEL
LIN {X 0,Y 268.501,Z 861.588,A -85,B 0,C 180,E1 18430.507,E2 18430.507} C_VEL
LIN {X 0,Y 255.096,Z 888.697,A -85,B 0,C 180,E1 18435.929,E2 18435.929} C_VEL
LIN {X 0,Y 242.96,Z 910.955,A -85,B 0,C 180,E1 18442.452,E2 18442.452} C_VEL
LIN {X 0,Y 232.981,Z 928.445,A -85,B 0,C 180,E1 18450,E2 18450} C_VEL
LIN {X 0,Y 226.038,Z 941.44,A -85,B 0,C 180,E1 18458.64,E2 18458.64} C_VEL
LIN {X 0,Y 223.038,Z 948.096,A -85,B 0,C 180,E1 18465.702,E2 18465.702} C_VEL
LIN {X 0,Y 220.913,Z 952.195,A -85,B 0,C 180,E1 18474.196,E2 18474.196} C_VEL
LIN {X 0,Y 221.535,Z 952.246,A -85,B 0,C 180,E1 18483.021,E2 18483.021} C_VEL
LIN {X 0,Y 224.931,Z 947.863,A -85,B 0,C 180,E1 18492.136,E2 18492.136} C_VEL
LIN {X 0,Y 231.608,Z 938.246,A -85,B 0,C 180,E1 18501.431,E2 18501.431} C_VEL
LIN {X 0,Y 243.003,Z 922.289,A -85,B 0,C 180,E1 18510.388,E2 18510.388} C_VEL
LIN {X 0,Y 257.13,Z 901.724,A -85,B 0,C 180,E1 18517.648,E2 18517.648} C_VEL
LIN {X 0,Y 272.843,Z 876.448,A -85,B 0,C 180,E1 18523.535,E2 18523.535} C_VEL
LIN {X 0,Y 288.64,Z 846.755,A -85,B 0,C 180,E1 18528.144,E2 18528.144} C_VEL
LIN {X 0,Y 294.434,Z 833.35,A -85,B 0,C 180,E1 18529.823,E2 18529.823} C_VEL
LIN {X 0,Y 294.118,Z 815.202,A -85,B 0,C 180,E1 18535.242,E2 18535.242} C_VEL
LIN {X 0,Y 292.525,Z 802.351,A -85,B 0,C 180,E1 18540.762,E2 18540.762} C_VEL
LIN {X 0,Y 291.528,Z 795.249,A -85,B 0,C 180,E1 18545.965,E2 18545.965} C_VEL
LIN {X 0,Y 291.242,Z 793.839,A -85,B 0,C 180,E1 18550.113,E2 18550.113} C_VEL
LIN {X 0,Y 291.69,Z 794.804,A -85,B 0,C 180,E1 18553.37,E2 18553.37} C_VEL
LIN {X 0,Y 293.952,Z 802.651,A -85,B 0,C 180,E1 18559.631,E2 18559.631} C_VEL
LIN {X 0,Y 297.365,Z 816.517,A -85,B 0,C 180,E1 18565.442,E2 18565.442} C_VEL
LIN {X 0,Y 299.806,Z 832.027,A -85,B 0,C 180,E1 18569.902,E2 18569.902} C_VEL
LIN {X 0,Y 299.571,Z 837.854,A -85,B 0,C 180,E1 18571.091,E2 18571.091} C_VEL
LIN {X 0,Y 284.337,Z 872.436,A -85,B 0,C 180,E1 18574.652,E2 18574.652} C_VEL
LIN {X 0,Y 268.259,Z 902.935,A -85,B 0,C 180,E1 18579.333,E2 18579.333} C_VEL
LIN {X 0,Y 252.033,Z 930.447,A -85,B 0,C 180,E1 18585.581,E2 18585.581} C_VEL
LIN {X 0,Y 237.158,Z 954.833,A -85,B 0,C 180,E1 18593.967,E2 18593.967} C_VEL
LIN {X 0,Y 227.086,Z 973.001,A -85,B 0,C 180,E1 18603.577,E2 18603.577} C_VEL
LIN {X 0,Y 222.597,Z 984.213,A -85,B 0,C 180,E1 18612.799,E2 18612.799} C_VEL
LIN {X 0,Y 221.342,Z 990.671,A -85,B 0,C 180,E1 18622.163,E2 18622.163} C_VEL
LIN {X 0,Y 221.811,Z 992.307,A -85,B 0,C 180,E1 18629.999,E2 18629.999} C_VEL
LIN {X 0,Y 221.366,Z 989.605,A -85,B 0,C 180,E1 18639.322,E2 18639.322} C_VEL
LIN {X 0,Y 223.116,Z 981.821,A -85,B 0,C 180,E1 18648.703,E2 18648.703} C_VEL
LIN {X 0,Y 228.788,Z 967.703,A -85,B 0,C 180,E1 18658.567,E2 18658.567} C_VEL
LIN {X 0,Y 238.77,Z 948.167,A -85,B 0,C 180,E1 18667.343,E2 18667.343} C_VEL
LIN {X 0,Y 251.884,Z 923.878,A -85,B 0,C 180,E1 18674.648,E2 18674.648} C_VEL
LIN {X 0,Y 266.397,Z 895.19,A -85,B 0,C 180,E1 18680.515,E2 18680.515} C_VEL
LIN {X 0,Y 280.872,Z 862.568,A -85,B 0,C 180,E1 18685.014,E2 18685.014} C_VEL
LIN {X 0,Y 291.446,Z 832.813,A -85,B 0,C 180,E1 18687.927,E2 18687.927} C_VEL
LIN {X 0,Y 283.901,Z 806.412,A -85,B 0,C 180,E1 18693.758,E2 18693.758} C_VEL
LIN {X 0,Y 273.443,Z 780.983,A -85,B 0,C 180,E1 18700.576,E2 18700.576} C_VEL
LIN {X 0,Y 263.478,Z 762.337,A -85,B 0,C 180,E1 18707.201,E2 18707.201} C_VEL
LIN {X 0,Y 254.237,Z 746.535,A -85,B 0,C 180,E1 18714.652,E2 18714.652} C_VEL
LIN {X 0,Y 249.207,Z 739.19,A -85,B 0,C 180,E1 18719.755,E2 18719.755} C_VEL
LIN {X 0,Y 245.579,Z 733.344,A -85,B 0,C 180,E1 18724.817,E2 18724.817} C_VEL
LIN {X 0,Y 244.357,Z 732.794,A -85,B 0,C 180,E1 18726.787,E2 18726.787} C_VEL
LIN {X 0,Y 241.905,Z 735.663,A -85,B 0,C 180,E1 18730.825,E2 18730.825} C_VEL
LIN {X 0,Y 240.341,Z 738.968,A -85,B 0,C 180,E1 18734.925,E2 18734.925} C_VEL
LIN {X 0,Y 242.554,Z 741.486,A -85,B 0,C 180,E1 18747.244,E2 18747.244} C_VEL
LIN {X 0,Y 246.345,Z 747.918,A -85,B 0,C 180,E1 18753.725,E2 18753.725} C_VEL
LIN {X 0,Y 252.426,Z 759.022,A -85,B 0,C 180,E1 18760.948,E2 18760.948} C_VEL
LIN {X 0,Y 259.606,Z 772.245,A -85,B 0,C 180,E1 18767.536,E2 18767.536} C_VEL
LIN {X 0,Y 267.702,Z 790.945,A -85,B 0,C 180,E1 18774.378,E2 18774.378} C_VEL
LIN {X 0,Y 273.882,Z 811.14,A -85,B 0,C 180,E1 18780.273,E2 18780.273} C_VEL
LIN {X 0,Y 276.979,Z 829.257,A -85,B 0,C 180,E1 18784.845,E2 18784.845} C_VEL
LIN {X 0,Y 263.127,Z 861.634,A -85,B 0,C 180,E1 18789.216,E2 18789.216} C_VEL
LIN {X 0,Y 248.759,Z 889.651,A -85,B 0,C 180,E1 18794.882,E2 18794.882} C_VEL
LIN {X 0,Y 235.678,Z 912.574,A -85,B 0,C 180,E1 18801.792,E2 18801.792} C_VEL
LIN {X 0,Y 224.92,Z 930.632,A -85,B 0,C 180,E1 18810.001,E2 18810.001} C_VEL
LIN {X 0,Y 217.966,Z 943.141,A -85,B 0,C 180,E1 18818.962,E2 18818.962} C_VEL
LIN {X 0,Y 214.893,Z 949.371,A -85,B 0,C 180,E1 18826.314,E2 18826.314} C_VEL
LIN {X 0,Y 212.98,Z 953.122,A -85,B 0,C 180,E1 18835.159,E2 18835.159} C_VEL
LIN {X 0,Y 214.008,Z 952.784,A -85,B 0,C 180,E1 18844.341,E2 18844.341} C_VEL
LIN {X 0,Y 217.903,Z 947.914,A -85,B 0,C 180,E1 18853.831,E2 18853.831} C_VEL
LIN {X 0,Y 225.55,Z 937.702,A -85,B 0,C 180,E1 18863.404,E2 18863.404} C_VEL
LIN {X 0,Y 237.335,Z 922.216,A -85,B 0,C 180,E1 18871.975,E2 18871.975} C_VEL
LIN {X 0,Y 252.21,Z 901.709,A -85,B 0,C 180,E1 18879.206,E2 18879.206} C_VEL
LIN {X 0,Y 268.807,Z 876.14,A -85,B 0,C 180,E1 18885.108,E2 18885.108} C_VEL
LIN {X 0,Y 286.031,Z 844.543,A -85,B 0,C 180,E1 18889.878,E2 18889.878} C_VEL
LIN {X 0,Y 289.434,Z 836.419,A -85,B 0,C 180,E1 18891.028,E2 18891.028} C_VEL
LIN {X 0,Y 289.693,Z 819.826,A -85,B 0,C 180,E1 18896.292,E2 18896.292} C_VEL
LIN {X 0,Y 288.785,Z 807.312,A -85,B 0,C 180,E1 18902.205,E2 18902.205} C_VEL
LIN {X 0,Y 288.376,Z 802.444,A -85,B 0,C 180,E1 18906.148,E2 18906.148} C_VEL
LIN {X 0,Y 288.312,Z 801.085,A -85,B 0,C 180,E1 18909.056,E2 18909.056} C_VEL
LIN {X 0,Y 288.695,Z 802.548,A -85,B 0,C 180,E1 18913.626,E2 18913.626} C_VEL
LIN {X 0,Y 290.623,Z 810.372,A -85,B 0,C 180,E1 18919.747,E2 18919.747} C_VEL
LIN {X 0,Y 293.399,Z 824.396,A -85,B 0,C 180,E1 18925.535,E2 18925.535} C_VEL
LIN {X 0,Y 294.904,Z 839.07,A -85,B 0,C 180,E1 18929.74,E2 18929.74} C_VEL
LIN {X 0,Y 278.614,Z 874.948,A -85,B 0,C 180,E1 18933.618,E2 18933.618} C_VEL
LIN {X 0,Y 260.968,Z 906.433,A -85,B 0,C 180,E1 18938.681,E2 18938.681} C_VEL
LIN {X 0,Y 243.979,Z 933.512,A -85,B 0,C 180,E1 18945.264,E2 18945.264} C_VEL
LIN {X 0,Y 229.221,Z 956.301,A -85,B 0,C 180,E1 18953.665,E2 18953.665} C_VEL
LIN {X 0,Y 219.071,Z 973.802,A -85,B 0,C 180,E1 18963.614,E2 18963.614} C_VEL
LIN {X 0,Y 214.457,Z 984.829,A -85,B 0,C 180,E1 18973.652,E2 18973.652} C_VEL
LIN {X 0,Y 213.479,Z 989.989,A -85,B 0,C 180,E1 18981.872,E2 18981.872} C_VEL
LIN {X 0,Y 213.949,Z 991.59,A -85,B 0,C 180,E1 18989.999,E2 18989.999} C_VEL
LIN {X 0,Y 213.478,Z 989.559,A -85,B 0,C 180,E1 18998.127,E2 18998.127} C_VEL
LIN {X 0,Y 214.89,Z 982.652,A -85,B 0,C 180,E1 19007.715,E2 19007.715} C_VEL
LIN {X 0,Y 220.215,Z 969.412,A -85,B 0,C 180,E1 19017.974,E2 19017.974} C_VEL
LIN {X 0,Y 229.948,Z 951.088,A -85,B 0,C 180,E1 19027.009,E2 19027.009} C_VEL
LIN {X 0,Y 243.872,Z 926.587,A -85,B 0,C 180,E1 19034.991,E2 19034.991} C_VEL
LIN {X 0,Y 259.59,Z 896.9,A -85,B 0,C 180,E1 19041.364,E2 19041.364} C_VEL
LIN {X 0,Y 274.528,Z 864.677,A -85,B 0,C 180,E1 19045.955,E2 19045.955} C_VEL
LIN {X 0,Y 285.362,Z 835.286,A -85,B 0,C 180,E1 19048.981,E2 19048.981} C_VEL
LIN {X 0,Y 278.483,Z 810.147,A -85,B 0,C 180,E1 19054.811,E2 19054.811} C_VEL
LIN {X 0,Y 269.555,Z 787.199,A -85,B 0,C 180,E1 19061.2,E2 19061.2} C_VEL
LIN {X 0,Y 260.049,Z 768.304,A -85,B 0,C 180,E1 19068.123,E2 19068.123} C_VEL
LIN {X 0,Y 251.899,Z 753.712,A -85,B 0,C 180,E1 19075.249,E2 19075.249} C_VEL
LIN {X 0,Y 247.239,Z 746.555,A -85,B 0,C 180,E1 19080.339,E2 19080.339} C_VEL
LIN {X 0,Y 243.896,Z 740.991,A -85,B 0,C 180,E1 19085.473,E2 19085.473} C_VEL
LIN {X 0,Y 240.341,Z 738.968,A -85,B 0,C 180,E1 19094.925,E2 19094.925} C_VEL
LIN {X 0,Y 239.683,Z 741.714,A -85,B 0,C 180,E1 19097.994,E2 19097.994} C_VEL
LIN {X 0,Y 239.209,Z 747.747,A -85,B 0,C 180,E1 19102.536,E2 19102.536} C_VEL
LIN {X 0,Y 239.322,Z 747.955,A -85,B 0,C 180,E1 19103.062,E2 19103.062} C_VEL
LIN {X 0,Y 240.913,Z 749.914,A -85,B 0,C 180,E1 19107.419,E2 19107.419} C_VEL
LIN {X 0,Y 244.927,Z 757.509,A -85,B 0,C 180,E1 19114.734,E2 19114.734} C_VEL
LIN {X 0,Y 250.741,Z 767.944,A -85,B 0,C 180,E1 19121.674,E2 19121.674} C_VEL
LIN {X 0,Y 258.493,Z 784.487,A -85,B 0,C 180,E1 19129.311,E2 19129.311} C_VEL
LIN {X 0,Y 265.797,Z 804.976,A -85,B 0,C 180,E1 19136.396,E2 19136.396} C_VEL
LIN {X 0,Y 270.228,Z 825.635,A -85,B 0,C 180,E1 19142.187,E2 19142.187} C_VEL
LIN {X 0,Y 270.777,Z 832.694,A -85,B 0,C 180,E1 19143.902,E2 19143.902} C_VEL
LIN {X 0,Y 256.321,Z 864.755,A -85,B 0,C 180,E1 19148.411,E2 19148.411} C_VEL
LIN {X 0,Y 241.856,Z 891.712,A -85,B 0,C 180,E1 19154.058,E2 19154.058} C_VEL
LIN {X 0,Y 228.175,Z 914.632,A -85,B 0,C 180,E1 19161.256,E2 19161.256} C_VEL
LIN {X 0,Y 216.833,Z 932.702,A -85,B 0,C 180,E1 19170.001,E2 19170.001} C_VEL
LIN {X 0,Y 209.899,Z 944.687,A -85,B 0,C 180,E1 19179.31,E2 19179.31} C_VEL
LIN {X 0,Y 206.384,Z 951.397,A -85,B 0,C 180,E1 19188.248,E2 19188.248} C_VEL
LIN {X 0,Y 205.018,Z 954.203,A -85,B 0,C 180,E1 19198.06,E2 19198.06} C_VEL
LIN {X 0,Y 206.816,Z 952.874,A -85,B 0,C 180,E1 19206.694,E2 19206.694} C_VEL
LIN {X 0,Y 212.066,Z 946.612,A -85,B 0,C 180,E1 19217.109,E2 19217.109} C_VEL
LIN {X 0,Y 221.843,Z 934.683,A -85,B 0,C 180,E1 19227.078,E2 19227.078} C_VEL
LIN {X 0,Y 236.106,Z 916.841,A -85,B 0,C 180,E1 19235.829,E2 19235.829} C_VEL
LIN {X 0,Y 252.769,Z 894.313,A -85,B 0,C 180,E1 19242.786,E2 19242.786} C_VEL
LIN {X 0,Y 270.734,Z 866.479,A -85,B 0,C 180,E1 19248.333,E2 19248.333} C_VEL
LIN {X 0,Y 284.332,Z 841.028,A -85,B 0,C 180,E1 19251.799,E2 19251.799} C_VEL
LIN {X 0,Y 285.317,Z 825.405,A -85,B 0,C 180,E1 19256.993,E2 19256.993} C_VEL
LIN {X 0,Y 285.108,Z 813.292,A -85,B 0,C 180,E1 19263.058,E2 19263.058} C_VEL
LIN {X 0,Y 285.067,Z 809.823,A -85,B 0,C 180,E1 19266.1,E2 19266.1} C_VEL
LIN {X 0,Y 285.079,Z 808.283,A -85,B 0,C 180,E1 19269.16,E2 19269.16} C_VEL
LIN {X 0,Y 285.294,Z 808.817,A -85,B 0,C 180,E1 19272.237,E2 19272.237} C_VEL
LIN {X 0,Y 286.753,Z 815.952,A -85,B 0,C 180,E1 19278.693,E2 19278.693} C_VEL
LIN {X 0,Y 288.779,Z 828.459,A -85,B 0,C 180,E1 19284.32,E2 19284.32} C_VEL
LIN {X 0,Y 289.86,Z 842.421,A -85,B 0,C 180,E1 19288.632,E2 19288.632} C_VEL
LIN {X 0,Y 272.819,Z 877.511,A -85,B 0,C 180,E1 19292.55,E2 19292.55} C_VEL
LIN {X 0,Y 254.826,Z 908.01,A -85,B 0,C 180,E1 19297.623,E2 19297.623} C_VEL
LIN {X 0,Y 237.855,Z 933.687,A -85,B 0,C 180,E1 19304.046,E2 19304.046} C_VEL
LIN {X 0,Y 222.681,Z 955.805,A -85,B 0,C 180,E1 19312.417,E2 19312.417} C_VEL
LIN {X 0,Y 211.733,Z 973.212,A -85,B 0,C 180,E1 19322.624,E2 19322.624} C_VEL
LIN {X 0,Y 206.702,Z 984.178,A -85,B 0,C 180,E1 19333.021,E2 19333.021} C_VEL
LIN {X 0,Y 205.581,Z 989.299,A -85,B 0,C 180,E1 19341.558,E2 19341.558} C_VEL
LIN {X 0,Y 206.091,Z 990.87,A -85,B 0,C 180,E1 19349.999,E2 19349.999} C_VEL
LIN {X 0,Y 205.592,Z 988.795,A -85,B 0,C 180,E1 19358.441,E2 19358.441} C_VEL
LIN {X 0,Y 207.288,Z 981.434,A -85,B 0,C 180,E1 19368.784,E2 19368.784} C_VEL
LIN {X 0,Y 212.57,Z 969.252,A -85,B 0,C 180,E1 19378.499,E2 19378.499} C_VEL
LIN {X 0,Y 222.462,Z 951.576,A -85,B 0,C 180,E1 19387.625,E2 19387.625} C_VEL
LIN {X 0,Y 236.434,Z 928.035,A -85,B 0,C 180,E1 19395.642,E2 19395.642} C_VEL
LIN {X 0,Y 251.721,Z 900.605,A -85,B 0,C 180,E1 19401.876,E2 19401.876} C_VEL
LIN {X 0,Y 268.035,Z 867.347,A -85,B 0,C 180,E1 19406.872,E2 19406.872} C_VEL
LIN {X 0,Y 279.456,Z 839.023,A -85,B 0,C 180,E1 19409.765,E2 19409.765} C_VEL
LIN {X 0,Y 272.965,Z 813.71,A -85,B 0,C 180,E1 19415.917,E2 19415.917} C_VEL
LIN {X 0,Y 265.056,Z 792.397,A -85,B 0,C 180,E1 19422.158,E2 19422.158} C_VEL
LIN {X 0,Y 255.93,Z 772.877,A -85,B 0,C 180,E1 19429.572,E2 19429.572} C_VEL
LIN {X 0,Y 248.464,Z 759.586,A -85,B 0,C 180,E1 19436.764,E2 19436.764} C_VEL
LIN {X 0,Y 245.173,Z 753.884,A -85,B 0,C 180,E1 19440.874,E2 19440.874} C_VEL
LIN {X 0,Y 242.174,Z 748.653,A -85,B 0,C 180,E1 19445.762,E2 19445.762} C_VEL
LIN {X 0,Y 238.825,Z 746.709,A -85,B 0,C 180,E1 19454.886,E2 19454.886} C_VEL
LIN {X 0,Y 239.322,Z 747.955,A -85,B 0,C 180,E1 19463.062,E2 19463.062} C_VEL
LIN {X 0,Y 239.698,Z 751.931,A -85,B 0,C 180,E1 19466.05,E2 19466.05} C_VEL
LIN {X 0,Y 240.145,Z 760.826,A -85,B 0,C 180,E1 19470.354,E2 19470.354} C_VEL
LIN {X 0,Y 240.394,Z 761.338,A -85,B 0,C 180,E1 19470.868,E2 19470.868} C_VEL
LIN {X 0,Y 242.529,Z 765.042,A -85,B 0,C 180,E1 19474.488,E2 19474.488} C_VEL
LIN {X 0,Y 247.189,Z 774.032,A -85,B 0,C 180,E1 19480.677,E2 19480.677} C_VEL
LIN {X 0,Y 254.347,Z 790.351,A -85,B 0,C 180,E1 19488.552,E2 19488.552} C_VEL
LIN {X 0,Y 260.692,Z 809.604,A -85,B 0,C 180,E1 19495.508,E2 19495.508} C_VEL
LIN {X 0,Y 264.585,Z 830.087,A -85,B 0,C 180,E1 19501.494,E2 19501.494} C_VEL
LIN {X 0,Y 264.769,Z 835.631,A -85,B 0,C 180,E1 19502.874,E2 19502.874} C_VEL
LIN {X 0,Y 250.097,Z 866.815,A -85,B 0,C 180,E1 19507.378,E2 19507.378} C_VEL
LIN {X 0,Y 234.973,Z 893.791,A -85,B 0,C 180,E1 19513.201,E2 19513.201} C_VEL
LIN {X 0,Y 220.606,Z 916.663,A -85,B 0,C 180,E1 19520.706,E2 19520.706} C_VEL
LIN {X 0,Y 208.728,Z 934.705,A -85,B 0,C 180,E1 19530.001,E2 19530.001} C_VEL
LIN {X 0,Y 201.466,Z 946.903,A -85,B 0,C 180,E1 19540.436,E2 19540.436} C_VEL
LIN {X 0,Y 198.667,Z 951.914,A -85,B 0,C 180,E1 19547.688,E2 19547.688} C_VEL
LIN {X 0,Y 197.153,Z 954.806,A -85,B 0,C 180,E1 19557.339,E2 19557.339} C_VEL
LIN {X 0,Y 199.156,Z 953.583,A -85,B 0,C 180,E1 19567.314,E2 19567.314} C_VEL
LIN {X 0,Y 204.434,Z 947.751,A -85,B 0,C 180,E1 19577.575,E2 19577.575} C_VEL
LIN {X 0,Y 214.383,Z 936.438,A -85,B 0,C 180,E1 19587.638,E2 19587.638} C_VEL
LIN {X 0,Y 229.706,Z 918.545,A -85,B 0,C 180,E1 19596.886,E2 19596.886} C_VEL
LIN {X 0,Y 247.472,Z 895.775,A -85,B 0,C 180,E1 19604.091,E2 19604.091} C_VEL
LIN {X 0,Y 265.217,Z 869.603,A -85,B 0,C 180,E1 19609.419,E2 19609.419} C_VEL
LIN {X 0,Y 279.185,Z 845.138,A -85,B 0,C 180,E1 19612.852,E2 19612.852} C_VEL
LIN {X 0,Y 280.929,Z 830.953,A -85,B 0,C 180,E1 19617.716,E2 19617.716} C_VEL
LIN {X 0,Y 281.373,Z 820.526,A -85,B 0,C 180,E1 19623.098,E2 19623.098} C_VEL
LIN {X 0,Y 281.472,Z 816.926,A -85,B 0,C 180,E1 19626.179,E2 19626.179} C_VEL
LIN {X 0,Y 281.662,Z 815.421,A -85,B 0,C 180,E1 19629.272,E2 19629.272} C_VEL
LIN {X 0,Y 281.864,Z 816.148,A -85,B 0,C 180,E1 19632.388,E2 19632.388} C_VEL
LIN {X 0,Y 283.015,Z 823.188,A -85,B 0,C 180,E1 19638.679,E2 19638.679} C_VEL
LIN {X 0,Y 284.525,Z 836.857,A -85,B 0,C 180,E1 19644.7,E2 19644.7} C_VEL
LIN {X 0,Y 284.755,Z 846.102,A -85,B 0,C 180,E1 19647.589,E2 19647.589} C_VEL
LIN {X 0,Y 267.24,Z 879.953,A -85,B 0,C 180,E1 19651.432,E2 19651.432} C_VEL
LIN {X 0,Y 248.784,Z 909.612,A -85,B 0,C 180,E1 19656.515,E2 19656.515} C_VEL
LIN {X 0,Y 231.05,Z 934.974,A -85,B 0,C 180,E1 19663.103,E2 19663.103} C_VEL
LIN {X 0,Y 214.769,Z 957.355,A -85,B 0,C 180,E1 19672.062,E2 19672.062} C_VEL
LIN {X 0,Y 203.518,Z 974.284,A -85,B 0,C 180,E1 19682.892,E2 19682.892} C_VEL
LIN {X 0,Y 198.981,Z 983.531,A -85,B 0,C 180,E1 19692.34,E2 19692.34} C_VEL
LIN {X 0,Y 197.704,Z 988.607,A -85,B 0,C 180,E1 19701.219,E2 19701.219} C_VEL
LIN {X 0,Y 198.225,Z 990.15,A -85,B 0,C 180,E1 19709.999,E2 19709.999} C_VEL
LIN {X 0,Y 197.715,Z 988.026,A -85,B 0,C 180,E1 19718.78,E2 19718.78} C_VEL
LIN {X 0,Y 199.023,Z 982.302,A -85,B 0,C 180,E1 19727.655,E2 19727.655} C_VEL
LIN {X 0,Y 204.746,Z 969.476,A -85,B 0,C 180,E1 19738.806,E2 19738.806} C_VEL
LIN {X 0,Y 215.246,Z 951.595,A -85,B 0,C 180,E1 19748.476,E2 19748.476} C_VEL
LIN {X 0,Y 229.175,Z 929.204,A -85,B 0,C 180,E1 19756.411,E2 19756.411} C_VEL
LIN {X 0,Y 244.804,Z 902.431,A -85,B 0,C 180,E1 19762.745,E2 19762.745} C_VEL
LIN {X 0,Y 261.103,Z 870.759,A -85,B 0,C 180,E1 19767.697,E2 19767.697} C_VEL
LIN {X 0,Y 273.365,Z 841.514,A -85,B 0,C 180,E1 19770.867,E2 19770.867} C_VEL
LIN {X 0,Y 267.841,Z 818.433,A -85,B 0,C 180,E1 19776.75,E2 19776.75} C_VEL
LIN {X 0,Y 260.578,Z 797.526,A -85,B 0,C 180,E1 19783.145,E2 19783.145} C_VEL
LIN {X 0,Y 252.198,Z 778.826,A -85,B 0,C 180,E1 19790.612,E2 19790.612} C_VEL
LIN {X 0,Y 245.851,Z 766.604,A -85,B 0,C 180,E1 19797.402,E2 19797.402} C_VEL
LIN {X 0,Y 242.781,Z 761.016,A -85,B 0,C 180,E1 19801.537,E2 19801.537} C_VEL
LIN {X 0,Y 240.476,Z 756.358,A -85,B 0,C 180,E1 19805.794,E2 19805.794} C_VEL
LIN {X 0,Y 236.929,Z 754.535,A -85,B 0,C 180,E1 19817.184,E2 19817.184} C_VEL
LIN {X 0,Y 238.817,Z 757.313,A -85,B 0,C 180,E1 19826.987,E2 19826.987} C_VEL
LIN {X 0,Y 240.394,Z 761.338,A -85,B 0,C 180,E1 19830.868,E2 19830.868} C_VEL
LIN {X 0,Y 240.646,Z 765.626,A -85,B 0,C 180,E1 19832.699,E2 19832.699} C_VEL
LIN {X 0,Y 240.545,Z 773.87,A -85,B 0,C 180,E1 19835.251,E2 19835.251} C_VEL
LIN {X 0,Y 240.725,Z 774.341,A -85,B 0,C 180,E1 19835.585,E2 19835.585} C_VEL
LIN {X 0,Y 246.543,Z 786.937,A -85,B 0,C 180,E1 19843.491,E2 19843.491} C_VEL
LIN {X 0,Y 252.687,Z 803.879,A -85,B 0,C 180,E1 19850.867,E2 19850.867} C_VEL
LIN {X 0,Y 257.136,Z 821.929,A -85,B 0,C 180,E1 19857.047,E2 19857.047} C_VEL
LIN {X 0,Y 259.066,Z 838.025,A -85,B 0,C 180,E1 19861.748,E2 19861.748} C_VEL
LIN {X 0,Y 243.369,Z 869.91,A -85,B 0,C 180,E1 19866.475,E2 19866.475} C_VEL
LIN {X 0,Y 227.378,Z 897.016,A -85,B 0,C 180,E1 19872.624,E2 19872.624} C_VEL
LIN {X 0,Y 213.075,Z 918.641,A -85,B 0,C 180,E1 19880.132,E2 19880.132} C_VEL
LIN {X 0,Y 201.913,Z 934.819,A -85,B 0,C 180,E1 19888.731,E2 19888.731} C_VEL
LIN {X 0,Y 194.259,Z 946.742,A -85,B 0,C 180,E1 19898.938,E2 19898.938} C_VEL
LIN {X 0,Y 190.478,Z 953.078,A -85,B 0,C 180,E1 19908.476,E2 19908.476} C_VEL
LIN {X 0,Y 189.306,Z 955.654,A -85,B 0,C 180,E1 19918.837,E2 19918.837} C_VEL
LIN {X 0,Y 191.865,Z 953.985,A -85,B 0,C 180,E1 19928.992,E2 19928.992} C_VEL
LIN {X 0,Y 198.035,Z 947.673,A -85,B 0,C 180,E1 19939.642,E2 19939.642} C_VEL
LIN {X 0,Y 209.288,Z 935.809,A -85,B 0,C 180,E1 19949.91,E2 19949.91} C_VEL
LIN {X 0,Y 224.935,Z 918.466,A -85,B 0,C 180,E1 19958.715,E2 19958.715} C_VEL
LIN {X 0,Y 243.579,Z 895.68,A -85,B 0,C 180,E1 19965.849,E2 19965.849} C_VEL
LIN {X 0,Y 262.34,Z 868.996,A -85,B 0,C 180,E1 19971.169,E2 19971.169} C_VEL
LIN {X 0,Y 274.773,Z 847.711,A -85,B 0,C 180,E1 19974.252,E2 19974.252} C_VEL
LIN {X 0,Y 276.627,Z 834.697,A -85,B 0,C 180,E1 19979.244,E2 19979.244} C_VEL
LIN {X 0,Y 277.523,Z 825.597,A -85,B 0,C 180,E1 19984.702,E2 19984.702} C_VEL
LIN {X 0,Y 278.11,Z 822.485,A -85,B 0,C 180,E1 19989.391,E2 19989.391} C_VEL
LIN {X 0,Y 278.391,Z 825.257,A -85,B 0,C 180,E1 19994.668,E2 19994.668} C_VEL
LIN {X 0,Y 279.186,Z 831.883,A -85,B 0,C 180,E1 19999.483,E2 19999.483} C_VEL
LIN {X 0,Y 279.899,Z 845.191,A -85,B 0,C 180,E1 20005.056,E2 20005.056} C_VEL
LIN {X 0,Y 279.455,Z 850.536,A -85,B 0,C 180,E1 20006.564,E2 20006.564} C_VEL
LIN {X 0,Y 259.949,Z 885.393,A -85,B 0,C 180,E1 20010.698,E2 20010.698} C_VEL
LIN {X 0,Y 240.495,Z 914.466,A -85,B 0,C 180,E1 20016.073,E2 20016.073} C_VEL
LIN {X 0,Y 221.57,Z 939.776,A -85,B 0,C 180,E1 20023.333,E2 20023.333} C_VEL
LIN {X 0,Y 205.482,Z 960.576,A -85,B 0,C 180,E1 20032.708,E2 20032.708} C_VEL
LIN {X 0,Y 195.025,Z 975.688,A -85,B 0,C 180,E1 20043.582,E2 20043.582} C_VEL
LIN {X 0,Y 190.67,Z 984.449,A -85,B 0,C 180,E1 20053.918,E2 20053.918} C_VEL
LIN {X 0,Y 189.818,Z 987.913,A -85,B 0,C 180,E1 20060.851,E2 20060.851} C_VEL
LIN {X 0,Y 190.36,Z 989.428,A -85,B 0,C 180,E1 20069.999,E2 20069.999} C_VEL
LIN {X 0,Y 189.837,Z 987.254,A -85,B 0,C 180,E1 20079.147,E2 20079.147} C_VEL
LIN {X 0,Y 191.442,Z 981.021,A -85,B 0,C 180,E1 20088.863,E2 20088.863} C_VEL
LIN {X 0,Y 197.456,Z 968.733,A -85,B 0,C 180,E1 20099.785,E2 20099.785} C_VEL
LIN {X 0,Y 208.839,Z 950.457,A -85,B 0,C 180,E1 20109.887,E2 20109.887} C_VEL
LIN {X 0,Y 223.53,Z 927.871,A -85,B 0,C 180,E1 20117.952,E2 20117.952} C_VEL
LIN {X 0,Y 239.961,Z 900.694,A -85,B 0,C 180,E1 20124.344,E2 20124.344} C_VEL
LIN {X 0,Y 256.759,Z 868.823,A -85,B 0,C 180,E1 20129.264,E2 20129.264} C_VEL
LIN {X 0,Y 267.329,Z 843.82,A -85,B 0,C 180,E1 20132.061,E2 20132.061} C_VEL
LIN {X 0,Y 262.297,Z 821.652,A -85,B 0,C 180,E1 20138.017,E2 20138.017} C_VEL
LIN {X 0,Y 255.22,Z 800.264,A -85,B 0,C 180,E1 20144.938,E2 20144.938} C_VEL
LIN {X 0,Y 247.347,Z 781.878,A -85,B 0,C 180,E1 20152.965,E2 20152.965} C_VEL
LIN {X 0,Y 241.206,Z 769.355,A -85,B 0,C 180,E1 20160.878,E2 20160.878} C_VEL
LIN {X 0,Y 238.236,Z 763.856,A -85,B 0,C 180,E1 20166.333,E2 20166.333} C_VEL
LIN {X 0,Y 235.122,Z 762.134,A -85,B 0,C 180,E1 20175.698,E2 20175.698} C_VEL
LIN {X 0,Y 236.627,Z 764.719,A -85,B 0,C 180,E1 20186.581,E2 20186.581} C_VEL
LIN {X 0,Y 239.525,Z 771.146,A -85,B 0,C 180,E1 20193.314,E2 20193.314} C_VEL
LIN {X 0,Y 240.725,Z 774.341,A -85,B 0,C 180,E1 20195.585,E2 20195.585} C_VEL
LIN {X 0,Y 241.754,Z 780.46,A -85,B 0,C 180,E1 20198.328,E2 20198.328} C_VEL
LIN {X 0,Y 242.336,Z 792.166,A -85,B 0,C 180,E1 20202.184,E2 20202.184} C_VEL
LIN {X 0,Y 242.663,Z 793.08,A -85,B 0,C 180,E1 20202.657,E2 20202.657} C_VEL
LIN {X 0,Y 248.103,Z 809.634,A -85,B 0,C 180,E1 20210.217,E2 20210.217} C_VEL
LIN {X 0,Y 251.805,Z 826.592,A -85,B 0,C 180,E1 20216.257,E2 20216.257} C_VEL
LIN {X 0,Y 253.278,Z 840.735,A -85,B 0,C 180,E1 20220.599,E2 20220.599} C_VEL
LIN {X 0,Y 236.756,Z 872.818,A -85,B 0,C 180,E1 20225.526,E2 20225.526} C_VEL
LIN {X 0,Y 220.799,Z 898.603,A -85,B 0,C 180,E1 20231.574,E2 20231.574} C_VEL
LIN {X 0,Y 206.002,Z 919.98,A -85,B 0,C 180,E1 20239.237,E2 20239.237} C_VEL
LIN {X 0,Y 193.55,Z 937.179,A -85,B 0,C 180,E1 20248.945,E2 20248.945} C_VEL
LIN {X 0,Y 186.128,Z 948.271,A -85,B 0,C 180,E1 20259.332,E2 20259.332} C_VEL
LIN {X 0,Y 182.315,Z 954.206,A -85,B 0,C 180,E1 20269.335,E2 20269.335} C_VEL
LIN {X 0,Y 181.527,Z 956.358,A -85,B 0,C 180,E1 20279.92,E2 20279.92} C_VEL
LIN {X 0,Y 184.774,Z 954.314,A -85,B 0,C 180,E1 20290.795,E2 20290.795} C_VEL
LIN {X 0,Y 191.881,Z 947.516,A -85,B 0,C 180,E1 20301.855,E2 20301.855} C_VEL
LIN {X 0,Y 204.487,Z 935.069,A -85,B 0,C 180,E1 20312.32,E2 20312.32} C_VEL
LIN {X 0,Y 221.525,Z 917.231,A -85,B 0,C 180,E1 20321.086,E2 20321.086} C_VEL
LIN {X 0,Y 241.762,Z 893.377,A -85,B 0,C 180,E1 20328.223,E2 20328.223} C_VEL
LIN {X 0,Y 261.504,Z 865.612,A -85,B 0,C 180,E1 20333.401,E2 20333.401} C_VEL
LIN {X 0,Y 269.784,Z 852.112,A -85,B 0,C 180,E1 20335.23,E2 20335.23} C_VEL
LIN {X 0,Y 272.286,Z 840.204,A -85,B 0,C 180,E1 20340.025,E2 20340.025} C_VEL
LIN {X 0,Y 273.524,Z 832.57,A -85,B 0,C 180,E1 20344.771,E2 20344.771} C_VEL
LIN {X 0,Y 274.251,Z 829.43,A -85,B 0,C 180,E1 20349.525,E2 20349.525} C_VEL
LIN {X 0,Y 274.432,Z 831.932,A -85,B 0,C 180,E1 20354.349,E2 20354.349} C_VEL
LIN {X 0,Y 274.982,Z 838.601,A -85,B 0,C 180,E1 20359.246,E2 20359.246} C_VEL
LIN {X 0,Y 274.993,Z 851.907,A -85,B 0,C 180,E1 20364.861,E2 20364.861} C_VEL
LIN {X 0,Y 272.973,Z 856.765,A -85,B 0,C 180,E1 20365.654,E2 20365.654} C_VEL
LIN {X 0,Y 253.897,Z 888.667,A -85,B 0,C 180,E1 20369.63,E2 20369.63} C_VEL
LIN {X 0,Y 233.444,Z 917.496,A -85,B 0,C 180,E1 20375.225,E2 20375.225} C_VEL
LIN {X 0,Y 213.91,Z 942.058,A -85,B 0,C 180,E1 20382.709,E2 20382.709} C_VEL
LIN {X 0,Y 196.611,Z 963.113,A -85,B 0,C 180,E1 20393.116,E2 20393.116} C_VEL
LIN {X 0,Y 186.707,Z 976.683,A -85,B 0,C 180,E1 20404.027,E2 20404.027} C_VEL
LIN {X 0,Y 182.414,Z 985.198,A -85,B 0,C 180,E1 20415.63,E2 20415.63} C_VEL
LIN {X 0,Y 181.889,Z 988.381,A -85,B 0,C 180,E1 20425.24,E2 20425.24} C_VEL
LIN {X 0,Y 182.491,Z 988.706,A -85,B 0,C 180,E1 20429.999,E2 20429.999} C_VEL
LIN {X 0,Y 181.994,Z 986.478,A -85,B 0,C 180,E1 20439.545,E2 20439.545} C_VEL
LIN {X 0,Y 184.022,Z 979.529,A -85,B 0,C 180,E1 20450.396,E2 20450.396} C_VEL
LIN {X 0,Y 190.378,Z 967.731,A -85,B 0,C 180,E1 20461.011,E2 20461.011} C_VEL
LIN {X 0,Y 202.578,Z 949.296,A -85,B 0,C 180,E1 20471.384,E2 20471.384} C_VEL
LIN {X 0,Y 218.053,Z 926.494,A -85,B 0,C 180,E1 20479.574,E2 20479.574} C_VEL
LIN {X 0,Y 234.791,Z 899.795,A -85,B 0,C 180,E1 20485.848,E2 20485.848} C_VEL
LIN {X 0,Y 251.973,Z 868.126,A -85,B 0,C 180,E1 20490.706,E2 20490.706} C_VEL
LIN {X 0,Y 261.32,Z 846.473,A -85,B 0,C 180,E1 20493.202,E2 20493.202} C_VEL
LIN {X 0,Y 256.751,Z 824.817,A -85,B 0,C 180,E1 20499.327,E2 20499.327} C_VEL
LIN {X 0,Y 250.644,Z 805.297,A -85,B 0,C 180,E1 20506.04,E2 20506.04} C_VEL
LIN {X 0,Y 243.681,Z 787.97,A -85,B 0,C 180,E1 20513.926,E2 20513.926} C_VEL
LIN {X 0,Y 238.182,Z 776.111,A -85,B 0,C 180,E1 20521.899,E2 20521.899} C_VEL
LIN {X 0,Y 235.791,Z 771.272,A -85,B 0,C 180,E1 20526.861,E2 20526.861} C_VEL
LIN {X 0,Y 232.862,Z 769.799,A -85,B 0,C 180,E1 20536.919,E2 20536.919} C_VEL
LIN {X 0,Y 234.272,Z 772.387,A -85,B 0,C 180,E1 20546.445,E2 20546.445} C_VEL
LIN {X 0,Y 236.979,Z 779.413,A -85,B 0,C 180,E1 20553.625,E2 20553.625} C_VEL
LIN {X 0,Y 241.378,Z 790.19,A -85,B 0,C 180,E1 20560.98,E2 20560.98} C_VEL
LIN {X 0,Y 242.663,Z 793.08,A -85,B 0,C 180,E1 20562.657,E2 20562.657} C_VEL
LIN {X 0,Y 243.466,Z 800.328,A -85,B 0,C 180,E1 20565.222,E2 20565.222} C_VEL
LIN {X 0,Y 243.325,Z 814.63,A -85,B 0,C 180,E1 20569.245,E2 20569.245} C_VEL
LIN {X 0,Y 246.539,Z 831.971,A -85,B 0,C 180,E1 20575.687,E2 20575.687} C_VEL
LIN {X 0,Y 247.338,Z 843.987,A -85,B 0,C 180,E1 20579.481,E2 20579.481} C_VEL
LIN {X 0,Y 230.743,Z 874.685,A -85,B 0,C 180,E1 20584.326,E2 20584.326} C_VEL
LIN {X 0,Y 214.285,Z 900.191,A -85,B 0,C 180,E1 20590.458,E2 20590.458} C_VEL
LIN {X 0,Y 198.694,Z 921.67,A -85,B 0,C 180,E1 20598.444,E2 20598.444} C_VEL
LIN {X 0,Y 185.513,Z 939.042,A -85,B 0,C 180,E1 20608.835,E2 20608.835} C_VEL
LIN {X 0,Y 177.982,Z 949.761,A -85,B 0,C 180,E1 20619.764,E2 20619.764} C_VEL
LIN {X 0,Y 174.188,Z 955.332,A -85,B 0,C 180,E1 20630.276,E2 20630.276} C_VEL
LIN {X 0,Y 173.825,Z 957.06,A -85,B 0,C 180,E1 20641.392,E2 20641.392} C_VEL
LIN {X 0,Y 177.731,Z 954.583,A -85,B 0,C 180,E1 20652.785,E2 20652.785} C_VEL
LIN {X 0,Y 186.024,Z 947.306,A -85,B 0,C 180,E1 20664.214,E2 20664.214} C_VEL
LIN {X 0,Y 200.086,Z 934.364,A -85,B 0,C 180,E1 20674.828,E2 20674.828} C_VEL
LIN {X 0,Y 218.548,Z 916.034,A -85,B 0,C 180,E1 20683.517,E2 20683.517} C_VEL
LIN {X 0,Y 239.899,Z 891.506,A -85,B 0,C 180,E1 20690.482,E2 20690.482} C_VEL
LIN {X 0,Y 259.821,Z 864.145,A -85,B 0,C 180,E1 20695.341,E2 20695.341} C_VEL
LIN {X 0,Y 265.482,Z 854.854,A -85,B 0,C 180,E1 20696.768,E2 20696.768} C_VEL
LIN {X 0,Y 268.148,Z 844.136,A -85,B 0,C 180,E1 20701.638,E2 20701.638} C_VEL
LIN {X 0,Y 269.692,Z 837.719,A -85,B 0,C 180,E1 20706.45,E2 20706.45} C_VEL
LIN {X 0,Y 270.269,Z 836.307,A -85,B 0,C 180,E1 20709.666,E2 20709.666} C_VEL
LIN {X 0,Y 270.364,Z 839.051,A -85,B 0,C 180,E1 20714.569,E2 20714.569} C_VEL
LIN {X 0,Y 270.52,Z 845.229,A -85,B 0,C 180,E1 20719.041,E2 20719.041} C_VEL
LIN {X 0,Y 270.037,Z 856.322,A -85,B 0,C 180,E1 20723.922,E2 20723.922} C_VEL
LIN {X 0,Y 249.334,Z 889.934,A -85,B 0,C 180,E1 20728.193,E2 20728.193} C_VEL
LIN {X 0,Y 227.665,Z 918.95,A -85,B 0,C 180,E1 20733.933,E2 20733.933} C_VEL
LIN {X 0,Y 206.294,Z 944.139,A -85,B 0,C 180,E1 20742.02,E2 20742.02} C_VEL
LIN {X 0,Y 189.243,Z 963.606,A -85,B 0,C 180,E1 20752.292,E2 20752.292} C_VEL
LIN {X 0,Y 179.295,Z 976.222,A -85,B 0,C 180,E1 20763.034,E2 20763.034} C_VEL
LIN {X 0,Y 174.611,Z 984.539,A -85,B 0,C 180,E1 20774.973,E2 20774.973} C_VEL
LIN {X 0,Y 174.002,Z 987.674,A -85,B 0,C 180,E1 20785.024,E2 20785.024} C_VEL
LIN {X 0,Y 174.597,Z 987.98,A -85,B 0,C 180,E1 20789.999,E2 20789.999} C_VEL
LIN {X 0,Y 174.123,Z 985.695,A -85,B 0,C 180,E1 20799.981,E2 20799.981} C_VEL
LIN {X 0,Y 176.429,Z 978.643,A -85,B 0,C 180,E1 20811.315,E2 20811.315} C_VEL
LIN {X 0,Y 183.371,Z 966.706,A -85,B 0,C 180,E1 20822.337,E2 20822.337} C_VEL
LIN {X 0,Y 196.443,Z 948.106,A -85,B 0,C 180,E1 20832.98,E2 20832.98} C_VEL
LIN {X 0,Y 212.761,Z 925.098,A -85,B 0,C 180,E1 20841.276,E2 20841.276} C_VEL
LIN {X 0,Y 231.512,Z 896.096,A -85,B 0,C 180,E1 20847.925,E2 20847.925} C_VEL
LIN {X 0,Y 249.252,Z 863.511,A -85,B 0,C 180,E1 20852.667,E2 20852.667} C_VEL
LIN {X 0,Y 255.39,Z 849.373,A -85,B 0,C 180,E1 20854.314,E2 20854.314} C_VEL
LIN {X 0,Y 250.941,Z 826.696,A -85,B 0,C 180,E1 20861.103,E2 20861.103} C_VEL
LIN {X 0,Y 245.743,Z 809.144,A -85,B 0,C 180,E1 20867.563,E2 20867.563} C_VEL
LIN {X 0,Y 239.628,Z 793.127,A -85,B 0,C 180,E1 20875.458,E2 20875.458} C_VEL
LIN {X 0,Y 235.744,Z 783.746,A -85,B 0,C 180,E1 20881.804,E2 20881.804} C_VEL
LIN {X 0,Y 233.195,Z 778.728,A -85,B 0,C 180,E1 20887.404,E2 20887.404} C_VEL
LIN {X 0,Y 230.547,Z 777.486,A -85,B 0,C 180,E1 20899.067,E2 20899.067} C_VEL
LIN {X 0,Y 231.619,Z 779.408,A -85,B 0,C 180,E1 20905.816,E2 20905.816} C_VEL
LIN {X 0,Y 233.932,Z 786.227,A -85,B 0,C 180,E1 20913.009,E2 20913.009} C_VEL
LIN {X 0,Y 238.006,Z 797.595,A -85,B 0,C 180,E1 20920.887,E2 20920.887} C_VEL
LIN {X 0,Y 242.684,Z 812.093,A -85,B 0,C 180,E1 20928.201,E2 20928.201} C_VEL
LIN {X 0,Y 243.325,Z 814.63,A -85,B 0,C 180,E1 20929.245,E2 20929.245} C_VEL
LIN {X 0,Y 243.226,Z 822.961,A -85,B 0,C 180,E1 20931.64,E2 20931.64} C_VEL
LIN {X 0,Y 241.285,Z 838.184,A -85,B 0,C 180,E1 20935.445,E2 20935.445} C_VEL
LIN {X 0,Y 241.154,Z 847.597,A -85,B 0,C 180,E1 20938.382,E2 20938.382} C_VEL
LIN {X 0,Y 224.839,Z 876.492,A -85,B 0,C 180,E1 20943.062,E2 20943.062} C_VEL
LIN {X 0,Y 207.866,Z 901.733,A -85,B 0,C 180,E1 20949.274,E2 20949.274} C_VEL
LIN {X 0,Y 190.686,Z 924.253,A -85,B 0,C 180,E1 20958.011,E2 20958.011} C_VEL
LIN {X 0,Y 177.43,Z 940.839,A -85,B 0,C 180,E1 20968.782,E2 20968.782} C_VEL
LIN {X 0,Y 169.8,Z 951.136,A -85,B 0,C 180,E1 20980.239,E2 20980.239} C_VEL
LIN {X 0,Y 166.06,Z 956.432,A -85,B 0,C 180,E1 20991.315,E2 20991.315} C_VEL
LIN {X 0,Y 166.221,Z 957.772,A -85,B 0,C 180,E1 21003.005,E2 21003.005} C_VEL
LIN {X 0,Y 171.032,Z 954.768,A -85,B 0,C 180,E1 21015.173,E2 21015.173} C_VEL
LIN {X 0,Y 180.46,Z 947.12,A -85,B 0,C 180,E1 21026.743,E2 21026.743} C_VEL
LIN {X 0,Y 196.105,Z 933.695,A -85,B 0,C 180,E1 21037.43,E2 21037.43} C_VEL
LIN {X 0,Y 216.077,Z 914.607,A -85,B 0,C 180,E1 21046.052,E2 21046.052} C_VEL
LIN {X 0,Y 237.428,Z 890.908,A -85,B 0,C 180,E1 21052.511,E2 21052.511} C_VEL
LIN {X 0,Y 258.021,Z 863.433,A -85,B 0,C 180,E1 21057.195,E2 21057.195} C_VEL
LIN {X 0,Y 260.754,Z 859.338,A -85,B 0,C 180,E1 21057.769,E2 21057.769} C_VEL
LIN {X 0,Y 263.752,Z 849.589,A -85,B 0,C 180,E1 21062.485,E2 21062.485} C_VEL
LIN {X 0,Y 265.416,Z 844.464,A -85,B 0,C 180,E1 21066.554,E2 21066.554} C_VEL
LIN {X 0,Y 266.076,Z 843.101,A -85,B 0,C 180,E1 21069.82,E2 21069.82} C_VEL
LIN {X 0,Y 266.138,Z 846.741,A -85,B 0,C 180,E1 21075.437,E2 21075.437} C_VEL
LIN {X 0,Y 265.606,Z 855.47,A -85,B 0,C 180,E1 21080.703,E2 21080.703} C_VEL
LIN {X 0,Y 265.055,Z 860.65,A -85,B 0,C 180,E1 21082.84,E2 21082.84} C_VEL
LIN {X 0,Y 243.481,Z 893.126,A -85,B 0,C 180,E1 21087.01,E2 21087.01} C_VEL
LIN {X 0,Y 221.883,Z 920.418,A -85,B 0,C 180,E1 21092.613,E2 21092.613} C_VEL
LIN {X 0,Y 200.767,Z 943.982,A -85,B 0,C 180,E1 21100.36,E2 21100.36} C_VEL
LIN {X 0,Y 182.963,Z 962.931,A -85,B 0,C 180,E1 21110.567,E2 21110.567} C_VEL
LIN {X 0,Y 171.632,Z 976.175,A -85,B 0,C 180,E1 21122.437,E2 21122.437} C_VEL
LIN {X 0,Y 166.861,Z 983.874,A -85,B 0,C 180,E1 21134.257,E2 21134.257} C_VEL
LIN {X 0,Y 166.107,Z 986.971,A -85,B 0,C 180,E1 21144.787,E2 21144.787} C_VEL
LIN {X 0,Y 166.725,Z 987.254,A -85,B 0,C 180,E1 21149.999,E2 21149.999} C_VEL
LIN {X 0,Y 166.258,Z 984.906,A -85,B 0,C 180,E1 21160.458,E2 21160.458} C_VEL
LIN {X 0,Y 168.879,Z 977.737,A -85,B 0,C 180,E1 21172.318,E2 21172.318} C_VEL
LIN {X 0,Y 177.646,Z 964.033,A -85,B 0,C 180,E1 21184.986,E2 21184.986} C_VEL
LIN {X 0,Y 192.249,Z 944.546,A -85,B 0,C 180,E1 21195.745,E2 21195.745} C_VEL
LIN {X 0,Y 210.329,Z 919.848,A -85,B 0,C 180,E1 21204.11,E2 21204.11} C_VEL
LIN {X 0,Y 229.038,Z 891.226,A -85,B 0,C 180,E1 21210.224,E2 21210.224} C_VEL
LIN {X 0,Y 246.518,Z 859.267,A -85,B 0,C 180,E1 21214.603,E2 21214.603} C_VEL
LIN {X 0,Y 249.324,Z 853.542,A -85,B 0,C 180,E1 21215.212,E2 21215.212} C_VEL
LIN {X 0,Y 246.635,Z 835.122,A -85,B 0,C 180,E1 21220.775,E2 21220.775} C_VEL
LIN {X 0,Y 241.823,Z 816.115,A -85,B 0,C 180,E1 21227.816,E2 21227.816} C_VEL
LIN {X 0,Y 236.537,Z 800.781,A -85,B 0,C 180,E1 21235.398,E2 21235.398} C_VEL
LIN {X 0,Y 232.065,Z 789.444,A -85,B 0,C 180,E1 21243.697,E2 21243.697} C_VEL
LIN {X 0,Y 230.554,Z 786.164,A -85,B 0,C 180,E1 21247.49,E2 21247.49} C_VEL
LIN {X 0,Y 228.194,Z 784.732,A -85,B 0,C 180,E1 21255.303,E2 21255.303} C_VEL
LIN {X 0,Y 228.873,Z 786.655,A -85,B 0,C 180,E1 21265.336,E2 21265.336} C_VEL
LIN {X 0,Y 230.676,Z 792.939,A -85,B 0,C 180,E1 21272.355,E2 21272.355} C_VEL
LIN {X 0,Y 234.082,Z 803.702,A -85,B 0,C 180,E1 21280.09,E2 21280.09} C_VEL
LIN {X 0,Y 237.798,Z 816.387,A -85,B 0,C 180,E1 21286.846,E2 21286.846} C_VEL
LIN {X 0,Y 240.84,Z 833.248,A -85,B 0,C 180,E1 21293.706,E2 21293.706} C_VEL
LIN {X 0,Y 241.285,Z 838.184,A -85,B 0,C 180,E1 21295.445,E2 21295.445} C_VEL
LIN {X 0,Y 239.379,Z 844.648,A -85,B 0,C 180,E1 21296.711,E2 21296.711} C_VEL
LIN {X 0,Y 231.862,Z 857.058,A -85,B 0,C 180,E1 21298.062,E2 21298.062} C_VEL
LIN {X 0,Y 214.163,Z 885.65,A -85,B 0,C 180,E1 21303.309,E2 21303.309} C_VEL
LIN {X 0,Y 196.153,Z 910.193,A -85,B 0,C 180,E1 21310.332,E2 21310.332} C_VEL
LIN {X 0,Y 180.289,Z 929.518,A -85,B 0,C 180,E1 21319.146,E2 21319.146} C_VEL
LIN {X 0,Y 168.209,Z 944.004,A -85,B 0,C 180,E1 21330.001,E2 21330.001} C_VEL
LIN {X 0,Y 161.614,Z 952.503,A -85,B 0,C 180,E1 21340.764,E2 21340.764} C_VEL
LIN {X 0,Y 157.969,Z 957.414,A -85,B 0,C 180,E1 21352.465,E2 21352.465} C_VEL
LIN {X 0,Y 158.709,Z 958.424,A -85,B 0,C 180,E1 21364.785,E2 21364.785} C_VEL
LIN {X 0,Y 164.295,Z 955.143,A -85,B 0,C 180,E1 21377.29,E2 21377.29} C_VEL
LIN {X 0,Y 176.543,Z 945.912,A -85,B 0,C 180,E1 21390.401,E2 21390.401} C_VEL
LIN {X 0,Y 194.696,Z 931.047,A -85,B 0,C 180,E1 21401.184,E2 21401.184} C_VEL
LIN {X 0,Y 216.64,Z 910.724,A -85,B 0,C 180,E1 21409.462,E2 21409.462} C_VEL
LIN {X 0,Y 239.165,Z 885.793,A -85,B 0,C 180,E1 21415.489,E2 21415.489} C_VEL
LIN {X 0,Y 255.824,Z 863.832,A -85,B 0,C 180,E1 21418.938,E2 21418.938} C_VEL
LIN {X 0,Y 258.826,Z 856.282,A -85,B 0,C 180,E1 21422.532,E2 21422.532} C_VEL
LIN {X 0,Y 260.904,Z 851.039,A -85,B 0,C 180,E1 21426.668,E2 21426.668} C_VEL
LIN {X 0,Y 261.649,Z 849.768,A -85,B 0,C 180,E1 21429.988,E2 21429.988} C_VEL
LIN {X 0,Y 261.57,Z 853.609,A -85,B 0,C 180,E1 21435.648,E2 21435.648} C_VEL
LIN {X 0,Y 260.417,Z 863.251,A -85,B 0,C 180,E1 21441.135,E2 21441.135} C_VEL
LIN {X 0,Y 258.213,Z 867.476,A -85,B 0,C 180,E1 21441.893,E2 21441.893} C_VEL
LIN {X 0,Y 235.554,Z 899.113,A -85,B 0,C 180,E1 21446.248,E2 21446.248} C_VEL
LIN {X 0,Y 210.95,Z 927.667,A -85,B 0,C 180,E1 21452.803,E2 21452.803} C_VEL
LIN {X 0,Y 188.972,Z 950.254,A -85,B 0,C 180,E1 21461.527,E2 21461.527} C_VEL
LIN {X 0,Y 172.493,Z 966.808,A -85,B 0,C 180,E1 21472.237,E2 21472.237} C_VEL
LIN {X 0,Y 161.956,Z 978.634,A -85,B 0,C 180,E1 21485.21,E2 21485.21} C_VEL
LIN {X 0,Y 158.313,Z 985.16,A -85,B 0,C 180,E1 21499.009,E2 21499.009} C_VEL
LIN {X 0,Y 158.852,Z 986.529,A -85,B 0,C 180,E1 21509.999,E2 21509.999} C_VEL
LIN {X 0,Y 158.4,Z 984.107,A -85,B 0,C 180,E1 21520.983,E2 21520.983} C_VEL
LIN {X 0,Y 162.01,Z 975.772,A -85,B 0,C 180,E1 21534.78,E2 21534.78} C_VEL
LIN {X 0,Y 172.27,Z 961.171,A -85,B 0,C 180,E1 21547.819,E2 21547.819} C_VEL
LIN {X 0,Y 187.554,Z 941.972,A -85,B 0,C 180,E1 21558.093,E2 21558.093} C_VEL
LIN {X 0,Y 206.195,Z 917.412,A -85,B 0,C 180,E1 21566.219,E2 21566.219} C_VEL
LIN {X 0,Y 225.618,Z 888.373,A -85,B 0,C 180,E1 21572.214,E2 21572.214} C_VEL
LIN {X 0,Y 243.092,Z 856.932,A -85,B 0,C 180,E1 21576.361,E2 21576.361} C_VEL
LIN {X 0,Y 242.531,Z 846.577,A -85,B 0,C 180,E1 21579.368,E2 21579.368} C_VEL
LIN {X 0,Y 238.791,Z 827.399,A -85,B 0,C 180,E1 21586.265,E2 21586.265} C_VEL
LIN {X 0,Y 234.281,Z 811.761,A -85,B 0,C 180,E1 21593.5,E2 21593.5} C_VEL
LIN {X 0,Y 230.089,Z 799.181,A -85,B 0,C 180,E1 21601.594,E2 21601.594} C_VEL
LIN {X 0,Y 227.751,Z 793.56,A -85,B 0,C 180,E1 21607.582,E2 21607.582} C_VEL
LIN {X 0,Y 225.426,Z 792.145,A -85,B 0,C 180,E1 21615.496,E2 21615.496} C_VEL
LIN {X 0,Y 225.892,Z 793.983,A -85,B 0,C 180,E1 21625.145,E2 21625.145} C_VEL
LIN {X 0,Y 228.054,Z 802.57,A -85,B 0,C 180,E1 21634.179,E2 21634.179} C_VEL
LIN {X 0,Y 231.449,Z 814.617,A -85,B 0,C 180,E1 21642.272,E2 21642.272} C_VEL
LIN {X 0,Y 234.377,Z 829.153,A -85,B 0,C 180,E1 21649.298,E2 21649.298} C_VEL
LIN {X 0,Y 235.935,Z 845.702,A -85,B 0,C 180,E1 21655.671,E2 21655.671} C_VEL
LIN {X 0,Y 235.497,Z 850.348,A -85,B 0,C 180,E1 21657.119,E2 21657.119} C_VEL
LIN {X 0,Y 231.862,Z 857.058,A -85,B 0,C 180,E1 21658.062,E2 21658.062} C_VEL
LIN {X 0,Y 221.8,Z 870.452,A -85,B 0,C 180,E1 21659.384,E2 21659.384} C_VEL
LIN {X 0,Y 211.279,Z 883.122,A -85,B 0,C 180,E1 21660.968,E2 21660.968} C_VEL
LIN {X 0,Y 191.907,Z 908.929,A -85,B 0,C 180,E1 21668.068,E2 21668.068} C_VEL
LIN {X 0,Y 175.815,Z 927.785,A -85,B 0,C 180,E1 21676.348,E2 21676.348} C_VEL
LIN {X 0,Y 162.347,Z 943.011,A -85,B 0,C 180,E1 21687.337,E2 21687.337} C_VEL
LIN {X 0,Y 154.807,Z 952.06,A -85,B 0,C 180,E1 21698.228,E2 21698.228} C_VEL
LIN {X 0,Y 151.204,Z 956.603,A -85,B 0,C 180,E1 21707.422,E2 21707.422} C_VEL
LIN {X 0,Y 149.997,Z 959.268,A -85,B 0,C 180,E1 21720.201,E2 21720.201} C_VEL
LIN {X 0,Y 154.047,Z 957.738,A -85,B 0,C 180,E1 21733.293,E2 21733.293} C_VEL
LIN {X 0,Y 163.756,Z 951.458,A -85,B 0,C 180,E1 21746.493,E2 21746.493} C_VEL
LIN {X 0,Y 180.953,Z 938.869,A -85,B 0,C 180,E1 21758.8,E2 21758.8} C_VEL
LIN {X 0,Y 200.934,Z 922.471,A -85,B 0,C 180,E1 21767.506,E2 21767.506} C_VEL
LIN {X 0,Y 223.385,Z 900.936,A -85,B 0,C 180,E1 21774.274,E2 21774.274} C_VEL
LIN {X 0,Y 245.78,Z 875.069,A -85,B 0,C 180,E1 21779.225,E2 21779.225} C_VEL
LIN {X 0,Y 251.895,Z 866.918,A -85,B 0,C 180,E1 21780.457,E2 21780.457} C_VEL
LIN {X 0,Y 255.375,Z 859.195,A -85,B 0,C 180,E1 21785.111,E2 21785.111} C_VEL
LIN {X 0,Y 256.226,Z 857.506,A -85,B 0,C 180,E1 21786.79,E2 21786.79} C_VEL
LIN {X 0,Y 257.115,Z 856.341,A -85,B 0,C 180,E1 21790.166,E2 21790.166} C_VEL
LIN {X 0,Y 256.896,Z 859.829,A -85,B 0,C 180,E1 21795.352,E2 21795.352} C_VEL
LIN {X 0,Y 255.615,Z 867.372,A -85,B 0,C 180,E1 21799.905,E2 21799.905} C_VEL
LIN {X 0,Y 252.974,Z 871.739,A -85,B 0,C 180,E1 21800.644,E2 21800.644} C_VEL
LIN {X 0,Y 230.759,Z 900.961,A -85,B 0,C 180,E1 21804.762,E2 21804.762} C_VEL
LIN {X 0,Y 206.798,Z 927.443,A -85,B 0,C 180,E1 21810.869,E2 21810.869} C_VEL
LIN {X 0,Y 183.646,Z 949.952,A -85,B 0,C 180,E1 21819.614,E2 21819.614} C_VEL
LIN {X 0,Y 164.572,Z 967.787,A -85,B 0,C 180,E1 21831.761,E2 21831.761} C_VEL
LIN {X 0,Y 153.219,Z 979.808,A -85,B 0,C 180,E1 21846.799,E2 21846.799} C_VEL
LIN {X 0,Y 150.461,Z 984.479,A -85,B 0,C 180,E1 21858.428,E2 21858.428} C_VEL
LIN {X 0,Y 150.966,Z 985.8,A -85,B 0,C 180,E1 21869.999,E2 21869.999} C_VEL
LIN {X 0,Y 150.584,Z 983.286,A -85,B 0,C 180,E1 21881.561,E2 21881.561} C_VEL
LIN {X 0,Y 154.619,Z 974.793,A -85,B 0,C 180,E1 21896.051,E2 21896.051} C_VEL
LIN {X 0,Y 164.369,Z 961.912,A -85,B 0,C 180,E1 21908.262,E2 21908.262} C_VEL
LIN {X 0,Y 181.069,Z 941.9,A -85,B 0,C 180,E1 21919.505,E2 21919.505} C_VEL
LIN {X 0,Y 200.479,Z 917.401,A -85,B 0,C 180,E1 21927.77,E2 21927.77} C_VEL
LIN {X 0,Y 220.601,Z 888.432,A -85,B 0,C 180,E1 21933.784,E2 21933.784} C_VEL
LIN {X 0,Y 237.713,Z 857.914,A -85,B 0,C 180,E1 21937.954,E2 21937.954} C_VEL
LIN {X 0,Y 235.006,Z 837.624,A -85,B 0,C 180,E1 21945.09,E2 21945.09} C_VEL
LIN {X 0,Y 231.097,Z 821.172,A -85,B 0,C 180,E1 21952.467,E2 21952.467} C_VEL
LIN {X 0,Y 227.494,Z 808.803,A -85,B 0,C 180,E1 21959.969,E2 21959.969} C_VEL
LIN {X 0,Y 224.762,Z 800.898,A -85,B 0,C 180,E1 21967.684,E2 21967.684} C_VEL
LIN {X 0,Y 222.259,Z 799.698,A -85,B 0,C 180,E1 21978.099,E2 21978.099} C_VEL
LIN {X 0,Y 222.645,Z 800.802,A -85,B 0,C 180,E1 21983.955,E2 21983.955} C_VEL
LIN {X 0,Y 224.123,Z 808.08,A -85,B 0,C 180,E1 21992.546,E2 21992.546} C_VEL
LIN {X 0,Y 226.931,Z 819.714,A -85,B 0,C 180,E1 22001.051,E2 22001.051} C_VEL
LIN {X 0,Y 229.276,Z 833.645,A -85,B 0,C 180,E1 22008.173,E2 22008.173} C_VEL
LIN {X 0,Y 230.294,Z 849.309,A -85,B 0,C 180,E1 22014.555,E2 22014.555} C_VEL
LIN {X 0,Y 229.561,Z 853.785,A -85,B 0,C 180,E1 22015.896,E2 22015.896} C_VEL
LIN {X 0,Y 211.279,Z 883.122,A -85,B 0,C 180,E1 22020.968,E2 22020.968} C_VEL
LIN {X 0,Y 200.355,Z 895.014,A -85,B 0,C 180,E1 22022.895,E2 22022.895} C_VEL
LIN {X 0,Y 189.27,Z 906.095,A -85,B 0,C 180,E1 22025.202,E2 22025.202} C_VEL
LIN {X 0,Y 169.888,Z 928,A -85,B 0,C 180,E1 22034.546,E2 22034.546} C_VEL
LIN {X 0,Y 155.48,Z 943.38,A -85,B 0,C 180,E1 22045.826,E2 22045.826} C_VEL
LIN {X 0,Y 146.675,Z 953.31,A -85,B 0,C 180,E1 22058.519,E2 22058.519} C_VEL
LIN {X 0,Y 142.968,Z 957.716,A -85,B 0,C 180,E1 22068.461,E2 22068.461} C_VEL
LIN {X 0,Y 142.336,Z 959.993,A -85,B 0,C 180,E1 22082.103,E2 22082.103} C_VEL
LIN {X 0,Y 147.342,Z 958.144,A -85,B 0,C 180,E1 22095.801,E2 22095.801} C_VEL
LIN {X 0,Y 158.216,Z 951.637,A -85,B 0,C 180,E1 22109.139,E2 22109.139} C_VEL
LIN {X 0,Y 175.759,Z 939.705,A -85,B 0,C 180,E1 22120.812,E2 22120.812} C_VEL
LIN {X 0,Y 197.301,Z 922.997,A -85,B 0,C 180,E1 22129.654,E2 22129.654} C_VEL
LIN {X 0,Y 220.823,Z 901.368,A -85,B 0,C 180,E1 22136.306,E2 22136.306} C_VEL
LIN {X 0,Y 244.161,Z 875.269,A -85,B 0,C 180,E1 22141.127,E2 22141.127} C_VEL
LIN {X 0,Y 247.448,Z 871.178,A -85,B 0,C 180,E1 22141.703,E2 22141.703} C_VEL
LIN {X 0,Y 250.366,Z 865.607,A -85,B 0,C 180,E1 22145.214,E2 22145.214} C_VEL
LIN {X 0,Y 251.407,Z 863.903,A -85,B 0,C 180,E1 22146.921,E2 22146.921} C_VEL
LIN {X 0,Y 252.325,Z 862.781,A -85,B 0,C 180,E1 22150.361,E2 22150.361} C_VEL
LIN {X 0,Y 251.887,Z 866.74,A -85,B 0,C 180,E1 22155.666,E2 22155.666} C_VEL
LIN {X 0,Y 250.856,Z 871.103,A -85,B 0,C 180,E1 22158.435,E2 22158.435} C_VEL
LIN {X 0,Y 248.87,Z 874.444,A -85,B 0,C 180,E1 22159.179,E2 22159.179} C_VEL
LIN {X 0,Y 224.752,Z 904.421,A -85,B 0,C 180,E1 22163.498,E2 22163.498} C_VEL
LIN {X 0,Y 198.607,Z 931.519,A -85,B 0,C 180,E1 22170.144,E2 22170.144} C_VEL
LIN {X 0,Y 175.197,Z 952.651,A -85,B 0,C 180,E1 22179.176,E2 22179.176} C_VEL
LIN {X 0,Y 156.066,Z 969.167,A -85,B 0,C 180,E1 22191.766,E2 22191.766} C_VEL
LIN {X 0,Y 145.774,Z 979.186,A -85,B 0,C 180,E1 22205.538,E2 22205.538} C_VEL
LIN {X 0,Y 142.599,Z 983.798,A -85,B 0,C 180,E1 22217.78,E2 22217.78} C_VEL
LIN {X 0,Y 143.086,Z 985.072,A -85,B 0,C 180,E1 22229.999,E2 22229.999} C_VEL
LIN {X 0,Y 142.744,Z 982.442,A -85,B 0,C 180,E1 22242.205,E2 22242.205} C_VEL
LIN {X 0,Y 146.545,Z 974.962,A -85,B 0,C 180,E1 22255.952,E2 22255.952} C_VEL
LIN {X 0,Y 157.833,Z 960.865,A -85,B 0,C 180,E1 22270.052,E2 22270.052} C_VEL
LIN {X 0,Y 175.639,Z 940.733,A -85,B 0,C 180,E1 22281.471,E2 22281.471} C_VEL
LIN {X 0,Y 195.885,Z 916.157,A -85,B 0,C 180,E1 22289.718,E2 22289.718} C_VEL
LIN {X 0,Y 216.443,Z 887.332,A -85,B 0,C 180,E1 22295.602,E2 22295.602} C_VEL
LIN {X 0,Y 231.922,Z 860.579,A -85,B 0,C 180,E1 22299.305,E2 22299.305} C_VEL
LIN {X 0,Y 229.651,Z 840.602,A -85,B 0,C 180,E1 22306.797,E2 22306.797} C_VEL
LIN {X 0,Y 226.325,Z 825.233,A -85,B 0,C 180,E1 22314.231,E2 22314.231} C_VEL
LIN {X 0,Y 223.149,Z 812.996,A -85,B 0,C 180,E1 22322.492,E2 22322.492} C_VEL
LIN {X 0,Y 221.499,Z 808.093,A -85,B 0,C 180,E1 22327.798,E2 22327.798} C_VEL
LIN {X 0,Y 219.255,Z 806.747,A -85,B 0,C 180,E1 22335.943,E2 22335.943} C_VEL
LIN {X 0,Y 219.391,Z 808.336,A -85,B 0,C 180,E1 22344.333,E2 22344.333} C_VEL
LIN {X 0,Y 220.608,Z 815.903,A -85,B 0,C 180,E1 22353.13,E2 22353.13} C_VEL
LIN {X 0,Y 222.993,Z 828.31,A -85,B 0,C 180,E1 22361.894,E2 22361.894} C_VEL
LIN {X 0,Y 224.611,Z 843.041,A -85,B 0,C 180,E1 22369.318,E2 22369.318} C_VEL
LIN {X 0,Y 224.646,Z 855.338,A -85,B 0,C 180,E1 22374.306,E2 22374.306} C_VEL
LIN {X 0,Y 205.2,Z 885.411,A -85,B 0,C 180,E1 22379.631,E2 22379.631} C_VEL
LIN {X 0,Y 189.27,Z 906.095,A -85,B 0,C 180,E1 22385.202,E2 22385.202} C_VEL
LIN {X 0,Y 178.091,Z 916.264,A -85,B 0,C 180,E1 22387.981,E2 22387.981} C_VEL
LIN {X 0,Y 166.824,Z 925.538,A -85,B 0,C 180,E1 22391.219,E2 22391.219} C_VEL
LIN {X 0,Y 149.888,Z 942.671,A -85,B 0,C 180,E1 22403.116,E2 22403.116} C_VEL
LIN {X 0,Y 139.799,Z 953.164,A -85,B 0,C 180,E1 22416.198,E2 22416.198} C_VEL
LIN {X 0,Y 134.759,Z 958.831,A -85,B 0,C 180,E1 22429.63,E2 22429.63} C_VEL
LIN {X 0,Y 134.752,Z 960.721,A -85,B 0,C 180,E1 22444.052,E2 22444.052} C_VEL
LIN {X 0,Y 140.904,Z 958.467,A -85,B 0,C 180,E1 22458.563,E2 22458.563} C_VEL
LIN {X 0,Y 153.426,Z 951.537,A -85,B 0,C 180,E1 22472.277,E2 22472.277} C_VEL
LIN {X 0,Y 172.792,Z 939.191,A -85,B 0,C 180,E1 22483.876,E2 22483.876} C_VEL
LIN {X 0,Y 197.639,Z 920.597,A -85,B 0,C 180,E1 22493.023,E2 22493.023} C_VEL
LIN {X 0,Y 223.792,Z 896.686,A -85,B 0,C 180,E1 22499.507,E2 22499.507} C_VEL
LIN {X 0,Y 243.237,Z 874.999,A -85,B 0,C 180,E1 22503.217,E2 22503.217} C_VEL
LIN {X 0,Y 246.319,Z 870.103,A -85,B 0,C 180,E1 22507.065,E2 22507.065} C_VEL
LIN {X 0,Y 247.377,Z 869.098,A -85,B 0,C 180,E1 22510.571,E2 22510.571} C_VEL
LIN {X 0,Y 246.788,Z 872.651,A -85,B 0,C 180,E1 22515.338,E2 22515.338} C_VEL
LIN {X 0,Y 245.524,Z 876.43,A -85,B 0,C 180,E1 22517.572,E2 22517.572} C_VEL
LIN {X 0,Y 220.52,Z 906.064,A -85,B 0,C 180,E1 22521.833,E2 22521.833} C_VEL
LIN {X 0,Y 193.708,Z 932.289,A -85,B 0,C 180,E1 22528.354,E2 22528.354} C_VEL
LIN {X 0,Y 168.397,Z 953.735,A -85,B 0,C 180,E1 22537.857,E2 22537.857} C_VEL
LIN {X 0,Y 149.489,Z 968.863,A -85,B 0,C 180,E1 22550.003,E2 22550.003} C_VEL
LIN {X 0,Y 138.377,Z 978.576,A -85,B 0,C 180,E1 22564.137,E2 22564.137} C_VEL
LIN {X 0,Y 134.752,Z 983.12,A -85,B 0,C 180,E1 22577.057,E2 22577.057} C_VEL
LIN {X 0,Y 135.203,Z 984.342,A -85,B 0,C 180,E1 22589.999,E2 22589.999} C_VEL
LIN {X 0,Y 134.915,Z 981.591,A -85,B 0,C 180,E1 22602.926,E2 22602.926} C_VEL
LIN {X 0,Y 139.946,Z 973.032,A -85,B 0,C 180,E1 22618.702,E2 22618.702} C_VEL
LIN {X 0,Y 152.307,Z 958.885,A -85,B 0,C 180,E1 22632.653,E2 22632.653} C_VEL
LIN {X 0,Y 170.521,Z 939.401,A -85,B 0,C 180,E1 22643.625,E2 22643.625} C_VEL
LIN {X 0,Y 191.525,Z 914.86,A -85,B 0,C 180,E1 22651.754,E2 22651.754} C_VEL
LIN {X 0,Y 213.16,Z 885.31,A -85,B 0,C 180,E1 22657.627,E2 22657.627} C_VEL
LIN {X 0,Y 226.197,Z 863.95,A -85,B 0,C 180,E1 22660.487,E2 22660.487} C_VEL
LIN {X 0,Y 224.499,Z 845.213,A -85,B 0,C 180,E1 22667.846,E2 22667.846} C_VEL
LIN {X 0,Y 221.885,Z 830.952,A -85,B 0,C 180,E1 22675.093,E2 22675.093} C_VEL
LIN {X 0,Y 219.394,Z 819.719,A -85,B 0,C 180,E1 22682.925,E2 22682.925} C_VEL
LIN {X 0,Y 218.106,Z 815.225,A -85,B 0,C 180,E1 22687.92,E2 22687.92} C_VEL
LIN {X 0,Y 215.879,Z 813.943,A -85,B 0,C 180,E1 22696.199,E2 22696.199} C_VEL
LIN {X 0,Y 215.848,Z 815.827,A -85,B 0,C 180,E1 22704.759,E2 22704.759} C_VEL
LIN {X 0,Y 216.862,Z 823.746,A -85,B 0,C 180,E1 22713.779,E2 22713.779} C_VEL
LIN {X 0,Y 218.478,Z 835.51,A -85,B 0,C 180,E1 22722.003,E2 22722.003} C_VEL
LIN {X 0,Y 219.379,Z 850.223,A -85,B 0,C 180,E1 22729.51,E2 22729.51} C_VEL
LIN {X 0,Y 218.857,Z 858.763,A -85,B 0,C 180,E1 22733.033,E2 22733.033} C_VEL
LIN {X 0,Y 199.733,Z 886.98,A -85,B 0,C 180,E1 22738.072,E2 22738.072} C_VEL
LIN {X 0,Y 179.507,Z 911.712,A -85,B 0,C 180,E1 22745.146,E2 22745.146} C_VEL
LIN {X 0,Y 166.824,Z 925.538,A -85,B 0,C 180,E1 22751.219,E2 22751.219} C_VEL
LIN {X 0,Y 155.722,Z 933.88,A -85,B 0,C 180,E1 22755.041,E2 22755.041} C_VEL
LIN {X 0,Y 145.249,Z 941.147,A -85,B 0,C 180,E1 22759.624,E2 22759.624} C_VEL
LIN {X 0,Y 133.372,Z 952.589,A -85,B 0,C 180,E1 22773.244,E2 22773.244} C_VEL
LIN {X 0,Y 128.567,Z 957.63,A -85,B 0,C 180,E1 22783.578,E2 22783.578} C_VEL
LIN {X 0,Y 126.141,Z 961.156,A -85,B 0,C 180,E1 22798.59,E2 22798.59} C_VEL
LIN {X 0,Y 130.253,Z 960.69,A -85,B 0,C 180,E1 22814.038,E2 22814.038} C_VEL
LIN {X 0,Y 141.077,Z 955.81,A -85,B 0,C 180,E1 22828.84,E2 22828.84} C_VEL
LIN {X 0,Y 161.219,Z 944.461,A -85,B 0,C 180,E1 22842.841,E2 22842.841} C_VEL
LIN {X 0,Y 186.325,Z 927.651,A -85,B 0,C 180,E1 22852.802,E2 22852.802} C_VEL
LIN {X 0,Y 213.299,Z 905.489,A -85,B 0,C 180,E1 22859.806,E2 22859.806} C_VEL
LIN {X 0,Y 238.835,Z 879.295,A -85,B 0,C 180,E1 22864.558,E2 22864.558} C_VEL
LIN {X 0,Y 241.111,Z 876.215,A -85,B 0,C 180,E1 22867.218,E2 22867.218} C_VEL
LIN {X 0,Y 242.311,Z 875.334,A -85,B 0,C 180,E1 22870.794,E2 22870.794} C_VEL
LIN {X 0,Y 241.178,Z 879.61,A -85,B 0,C 180,E1 22875.841,E2 22875.841} C_VEL
LIN {X 0,Y 233.085,Z 889.556,A -85,B 0,C 180,E1 22877.264,E2 22877.264} C_VEL
LIN {X 0,Y 207.445,Z 916.522,A -85,B 0,C 180,E1 22881.954,E2 22881.954} C_VEL
LIN {X 0,Y 180.994,Z 939.803,A -85,B 0,C 180,E1 22888.903,E2 22888.903} C_VEL
LIN {X 0,Y 156.053,Z 959.019,A -85,B 0,C 180,E1 22899.321,E2 22899.321} C_VEL
LIN {X 0,Y 137.898,Z 972.441,A -85,B 0,C 180,E1 22912.995,E2 22912.995} C_VEL
LIN {X 0,Y 128,Z 981.049,A -85,B 0,C 180,E1 22930.71,E2 22930.71} C_VEL
LIN {X 0,Y 126.565,Z 983.445,A -85,B 0,C 180,E1 22943.151,E2 22943.151} C_VEL
LIN {X 0,Y 127.315,Z 983.611,A -85,B 0,C 180,E1 22949.999,E2 22949.999} C_VEL
LIN {X 0,Y 127.107,Z 980.73,A -85,B 0,C 180,E1 22963.735,E2 22963.735} C_VEL
LIN {X 0,Y 132.697,Z 972.171,A -85,B 0,C 180,E1 22980.199,E2 22980.199} C_VEL
LIN {X 0,Y 146.366,Z 957.649,A -85,B 0,C 180,E1 22994.866,E2 22994.866} C_VEL
LIN {X 0,Y 166.059,Z 937.575,A -85,B 0,C 180,E1 23006.116,E2 23006.116} C_VEL
LIN {X 0,Y 187.711,Z 913.133,A -85,B 0,C 180,E1 23014.004,E2 23014.004} C_VEL
LIN {X 0,Y 210.109,Z 883.237,A -85,B 0,C 180,E1 23019.702,E2 23019.702} C_VEL
LIN {X 0,Y 220.384,Z 866.375,A -85,B 0,C 180,E1 23022.027,E2 23022.027} C_VEL
LIN {X 0,Y 219.195,Z 848.521,A -85,B 0,C 180,E1 23029.559,E2 23029.559} C_VEL
LIN {X 0,Y 217.119,Z 834.981,A -85,B 0,C 180,E1 23036.981,E2 23036.981} C_VEL
LIN {X 0,Y 215.396,Z 825.77,A -85,B 0,C 180,E1 23043.984,E2 23043.984} C_VEL
LIN {X 0,Y 214.018,Z 821.959,A -85,B 0,C 180,E1 23049.205,E2 23049.205} C_VEL
LIN {X 0,Y 212.296,Z 821.032,A -85,B 0,C 180,E1 23056.48,E2 23056.48} C_VEL
LIN {X 0,Y 212.146,Z 823.248,A -85,B 0,C 180,E1 23065.221,E2 23065.221} C_VEL
LIN {X 0,Y 212.742,Z 829.933,A -85,B 0,C 180,E1 23073.017,E2 23073.017} C_VEL
LIN {X 0,Y 213.739,Z 841.581,A -85,B 0,C 180,E1 23081.509,E2 23081.509} C_VEL
LIN {X 0,Y 213.986,Z 855.392,A -85,B 0,C 180,E1 23088.837,E2 23088.837} C_VEL
LIN {X 0,Y 212.82,Z 862.582,A -85,B 0,C 180,E1 23091.707,E2 23091.707} C_VEL
LIN {X 0,Y 191.654,Z 892.092,A -85,B 0,C 180,E1 23097.227,E2 23097.227} C_VEL
LIN {X 0,Y 169.871,Z 916.911,A -85,B 0,C 180,E1 23105.042,E2 23105.042} C_VEL
LIN {X 0,Y 150.651,Z 936.022,A -85,B 0,C 180,E1 23115.499,E2 23115.499} C_VEL
LIN {X 0,Y 145.249,Z 941.147,A -85,B 0,C 180,E1 23119.624,E2 23119.624} C_VEL
LIN {X 0,Y 135.488,Z 947.491,A -85,B 0,C 180,E1 23124.984,E2 23124.984} C_VEL
LIN {X 0,Y 126.501,Z 952.712,A -85,B 0,C 180,E1 23131.21,E2 23131.21} C_VEL
LIN {X 0,Y 120.267,Z 958.857,A -85,B 0,C 180,E1 23144.534,E2 23144.534} C_VEL
LIN {X 0,Y 118.4,Z 962.014,A -85,B 0,C 180,E1 23160.652,E2 23160.652} C_VEL
LIN {X 0,Y 123.718,Z 961.167,A -85,B 0,C 180,E1 23177.042,E2 23177.042} C_VEL
LIN {X 0,Y 136.307,Z 955.893,A -85,B 0,C 180,E1 23192.335,E2 23192.335} C_VEL
LIN {X 0,Y 156.18,Z 945.535,A -85,B 0,C 180,E1 23205.066,E2 23205.066} C_VEL
LIN {X 0,Y 181.848,Z 929.383,A -85,B 0,C 180,E1 23214.749,E2 23214.749} C_VEL
LIN {X 0,Y 210.109,Z 907.395,A -85,B 0,C 180,E1 23221.691,E2 23221.691} C_VEL
LIN {X 0,Y 234.583,Z 883.59,A -85,B 0,C 180,E1 23226.024,E2 23226.024} C_VEL
LIN {X 0,Y 235.719,Z 882.211,A -85,B 0,C 180,E1 23227.384,E2 23227.384} C_VEL
LIN {X 0,Y 236.947,Z 881.405,A -85,B 0,C 180,E1 23231.042,E2 23231.042} C_VEL
LIN {X 0,Y 235.944,Z 884.466,A -85,B 0,C 180,E1 23234.682,E2 23234.682} C_VEL
LIN {X 0,Y 207.748,Z 913.873,A -85,B 0,C 180,E1 23239.214,E2 23239.214} C_VEL
LIN {X 0,Y 178.598,Z 938.626,A -85,B 0,C 180,E1 23246.136,E2 23246.136} C_VEL
LIN {X 0,Y 153.36,Z 957.101,A -85,B 0,C 180,E1 23255.733,E2 23255.733} C_VEL
LIN {X 0,Y 131.443,Z 971.945,A -85,B 0,C 180,E1 23270.844,E2 23270.844} C_VEL
LIN {X 0,Y 120.828,Z 979.981,A -85,B 0,C 180,E1 23287.995,E2 23287.995} C_VEL
LIN {X 0,Y 118.654,Z 982.744,A -85,B 0,C 180,E1 23302.692,E2 23302.692} C_VEL
LIN {X 0,Y 119.424,Z 982.878,A -85,B 0,C 180,E1 23309.999,E2 23309.999} C_VEL
LIN {X 0,Y 119.327,Z 979.863,A -85,B 0,C 180,E1 23324.65,E2 23324.65} C_VEL
LIN {X 0,Y 125.179,Z 971.724,A -85,B 0,C 180,E1 23341.247,E2 23341.247} C_VEL
LIN {X 0,Y 139.624,Z 957.388,A -85,B 0,C 180,E1 23356.509,E2 23356.509} C_VEL
LIN {X 0,Y 160.203,Z 937.496,A -85,B 0,C 180,E1 23367.966,E2 23367.966} C_VEL
LIN {X 0,Y 182.103,Z 913.796,A -85,B 0,C 180,E1 23375.717,E2 23375.717} C_VEL
LIN {X 0,Y 205.115,Z 884.238,A -85,B 0,C 180,E1 23381.384,E2 23381.384} C_VEL
LIN {X 0,Y 214.687,Z 869.507,A -85,B 0,C 180,E1 23383.379,E2 23383.379} C_VEL
LIN {X 0,Y 214.05,Z 852.971,A -85,B 0,C 180,E1 23390.741,E2 23390.741} C_VEL
LIN {X 0,Y 212.377,Z 839.07,A -85,B 0,C 180,E1 23398.95,E2 23398.95} C_VEL
LIN {X 0,Y 211.056,Z 830.847,A -85,B 0,C 180,E1 23405.996,E2 23405.996} C_VEL
LIN {X 0,Y 210.643,Z 829.133,A -85,B 0,C 180,E1 23408.202,E2 23408.202} C_VEL
LIN {X 0,Y 208.465,Z 828.023,A -85,B 0,C 180,E1 23416.792,E2 23416.792} C_VEL
LIN {X 0,Y 208.201,Z 828.618,A -85,B 0,C 180,E1 23421.206,E2 23421.206} C_VEL
LIN {X 0,Y 208.258,Z 832.677,A -85,B 0,C 180,E1 23428.612,E2 23428.612} C_VEL
LIN {X 0,Y 208.626,Z 841.035,A -85,B 0,C 180,E1 23436.459,E2 23436.459} C_VEL
LIN {X 0,Y 208.876,Z 852.091,A -85,B 0,C 180,E1 23443.744,E2 23443.744} C_VEL
LIN {X 0,Y 208.093,Z 863.767,A -85,B 0,C 180,E1 23449.675,E2 23449.675} C_VEL
LIN {X 0,Y 204.738,Z 869.383,A -85,B 0,C 180,E1 23450.778,E2 23450.778} C_VEL
LIN {X 0,Y 183.912,Z 896.454,A -85,B 0,C 180,E1 23456.217,E2 23456.217} C_VEL
LIN {X 0,Y 162.665,Z 919.391,A -85,B 0,C 180,E1 23463.855,E2 23463.855} C_VEL
LIN {X 0,Y 142.856,Z 938.03,A -85,B 0,C 180,E1 23474.688,E2 23474.688} C_VEL
LIN {X 0,Y 127.336,Z 951.979,A -85,B 0,C 180,E1 23490.001,E2 23490.001} C_VEL
LIN {X 0,Y 126.501,Z 952.712,A -85,B 0,C 180,E1 23491.21,E2 23491.21} C_VEL
LIN {X 0,Y 120.884,Z 955.993,A -85,B 0,C 180,E1 23496.507,E2 23496.507} C_VEL
LIN {X 0,Y 111.76,Z 960.16,A -85,B 0,C 180,E1 23506.241,E2 23506.241} C_VEL
LIN {X 0,Y 111.27,Z 962.936,A -85,B 0,C 180,E1 23525.666,E2 23525.666} C_VEL
LIN {X 0,Y 119.992,Z 960.84,A -85,B 0,C 180,E1 23543.951,E2 23543.951} C_VEL
LIN {X 0,Y 136.998,Z 953.787,A -85,B 0,C 180,E1 23559.575,E2 23559.575} C_VEL
LIN {X 0,Y 161.329,Z 941.156,A -85,B 0,C 180,E1 23571.528,E2 23571.528} C_VEL
LIN {X 0,Y 190.16,Z 922.526,A -85,B 0,C 180,E1 23580.036,E2 23580.036} C_VEL
LIN {X 0,Y 219.161,Z 898.715,A -85,B 0,C 180,E1 23585.736,E2 23585.736} C_VEL
LIN {X 0,Y 230.119,Z 888.028,A -85,B 0,C 180,E1 23587.565,E2 23587.565} C_VEL
LIN {X 0,Y 231.333,Z 887.734,A -85,B 0,C 180,E1 23591.906,E2 23591.906} C_VEL
LIN {X 0,Y 230.713,Z 888.98,A -85,B 0,C 180,E1 23593.246,E2 23593.246} C_VEL
LIN {X 0,Y 203.489,Z 915.744,A -85,B 0,C 180,E1 23597.415,E2 23597.415} C_VEL
LIN {X 0,Y 173.672,Z 939.729,A -85,B 0,C 180,E1 23604.168,E2 23604.168} C_VEL
LIN {X 0,Y 146.227,Z 958.434,A -85,B 0,C 180,E1 23614.351,E2 23614.351} C_VEL
LIN {X 0,Y 125.17,Z 971.463,A -85,B 0,C 180,E1 23628.464,E2 23628.464} C_VEL
LIN {X 0,Y 113.349,Z 979.355,A -85,B 0,C 180,E1 23646.459,E2 23646.459} C_VEL
LIN {X 0,Y 110.747,Z 982.041,A -85,B 0,C 180,E1 23662.168,E2 23662.168} C_VEL
LIN {X 0,Y 111.527,Z 982.128,A -85,B 0,C 180,E1 23669.999,E2 23669.999} C_VEL
LIN {X 0,Y 111.574,Z 978.986,A -85,B 0,C 180,E1 23685.693,E2 23685.693} C_VEL
LIN {X 0,Y 118.263,Z 970.683,A -85,B 0,C 180,E1 23703.303,E2 23703.303} C_VEL
LIN {X 0,Y 134.525,Z 955.738,A -85,B 0,C 180,E1 23719.374,E2 23719.374} C_VEL
LIN {X 0,Y 155.955,Z 935.993,A -85,B 0,C 180,E1 23730.556,E2 23730.556} C_VEL
LIN {X 0,Y 180.365,Z 910.302,A -85,B 0,C 180,E1 23738.554,E2 23738.554} C_VEL
LIN {X 0,Y 204.191,Z 879.714,A -85,B 0,C 180,E1 23743.889,E2 23743.889} C_VEL
LIN {X 0,Y 209.04,Z 872.25,A -85,B 0,C 180,E1 23744.953,E2 23744.953} C_VEL
LIN {X 0,Y 208.791,Z 856.04,A -85,B 0,C 180,E1 23752.702,E2 23752.702} C_VEL
LIN {X 0,Y 207.633,Z 843.08,A -85,B 0,C 180,E1 23761.112,E2 23761.112} C_VEL
LIN {X 0,Y 206.676,Z 835.969,A -85,B 0,C 180,E1 23768.361,E2 23768.361} C_VEL
LIN {X 0,Y 204.51,Z 834.929,A -85,B 0,C 180,E1 23777.127,E2 23777.127} C_VEL
LIN {X 0,Y 204.032,Z 836.909,A -85,B 0,C 180,E1 23784.581,E2 23784.581} C_VEL
LIN {X 0,Y 204.01,Z 842.816,A -85,B 0,C 180,E1 23792.242,E2 23792.242} C_VEL
LIN {X 0,Y 203.883,Z 853.347,A -85,B 0,C 180,E1 23800.497,E2 23800.497} C_VEL
LIN {X 0,Y 202.792,Z 866.708,A -85,B 0,C 180,E1 23808.018,E2 23808.018} C_VEL
LIN {X 0,Y 200.426,Z 870.695,A -85,B 0,C 180,E1 23808.938,E2 23808.938} C_VEL
LIN {X 0,Y 177.708,Z 899.091,A -85,B 0,C 180,E1 23814.689,E2 23814.689} C_VEL
LIN {X 0,Y 154.577,Z 922.813,A -85,B 0,C 180,E1 23823.022,E2 23823.022} C_VEL
LIN {X 0,Y 135.248,Z 939.839,A -85,B 0,C 180,E1 23833.668,E2 23833.668} C_VEL
LIN {X 0,Y 120.664,Z 952.129,A -85,B 0,C 180,E1 23847.77,E2 23847.77} C_VEL
LIN {X 0,Y 113.844,Z 958.181,A -85,B 0,C 180,E1 23860.148,E2 23860.148} C_VEL
LIN {X 0,Y 111.76,Z 960.16,A -85,B 0,C 180,E1 23866.241,E2 23866.241} C_VEL
LIN {X 0,Y 107.962,Z 961.891,A -85,B 0,C 180,E1 23872.749,E2 23872.749} C_VEL
LIN {X 0,Y 102.932,Z 963.538,A -85,B 0,C 180,E1 23883.185,E2 23883.185} C_VEL
LIN {X 0,Y 103.072,Z 963.579,A -85,B 0,C 180,E1 23884.407,E2 23884.407} C_VEL
LIN {X 0,Y 111.767,Z 962.168,A -85,B 0,C 180,E1 23904.107,E2 23904.107} C_VEL
LIN {X 0,Y 128.451,Z 956.155,A -85,B 0,C 180,E1 23920.025,E2 23920.025} C_VEL
LIN {X 0,Y 152.33,Z 945.074,A -85,B 0,C 180,E1 23932.156,E2 23932.156} C_VEL
LIN {X 0,Y 181.104,Z 928.173,A -85,B 0,C 180,E1 23940.834,E2 23940.834} C_VEL
LIN {X 0,Y 210.911,Z 905.853,A -85,B 0,C 180,E1 23946.718,E2 23946.718} C_VEL
LIN {X 0,Y 224.388,Z 893.871,A -85,B 0,C 180,E1 23948.732,E2 23948.732} C_VEL
LIN {X 0,Y 225.797,Z 893.234,A -85,B 0,C 180,E1 23951.594,E2 23951.594} C_VEL
LIN {X 0,Y 194.01,Z 922.153,A -85,B 0,C 180,E1 23956.533,E2 23956.533} C_VEL
LIN {X 0,Y 164.416,Z 943.909,A -85,B 0,C 180,E1 23963.39,E2 23963.39} C_VEL
LIN {X 0,Y 135.207,Z 961.948,A -85,B 0,C 180,E1 23974.776,E2 23974.776} C_VEL
LIN {X 0,Y 113.2,Z 974.328,A -85,B 0,C 180,E1 23992.083,E2 23992.083} C_VEL
LIN {X 0,Y 103.628,Z 980.445,A -85,B 0,C 180,E1 24013.067,E2 24013.067} C_VEL
LIN {X 0,Y 103.619,Z 981.347,A -85,B 0,C 180,E1 24029.999,E2 24029.999} C_VEL
LIN {X 0,Y 103.843,Z 978.099,A -85,B 0,C 180,E1 24046.895,E2 24046.895} C_VEL
LIN {X 0,Y 111.507,Z 969.607,A -85,B 0,C 180,E1 24065.622,E2 24065.622} C_VEL
LIN {X 0,Y 126.948,Z 956.441,A -85,B 0,C 180,E1 24080.591,E2 24080.591} C_VEL
LIN {X 0,Y 149.262,Z 937.015,A -85,B 0,C 180,E1 24092.203,E2 24092.203} C_VEL
LIN {X 0,Y 172.904,Z 913.381,A -85,B 0,C 180,E1 24099.883,E2 24099.883} C_VEL
LIN {X 0,Y 197.015,Z 884.28,A -85,B 0,C 180,E1 24105.238,E2 24105.238} C_VEL
LIN {X 0,Y 203.386,Z 874.789,A -85,B 0,C 180,E1 24106.678,E2 24106.678} C_VEL
LIN {X 0,Y 203.668,Z 861.189,A -85,B 0,C 180,E1 24113.586,E2 24113.586} C_VEL
LIN {X 0,Y 203.065,Z 848.712,A -85,B 0,C 180,E1 24122.095,E2 24122.095} C_VEL
LIN {X 0,Y 202.427,Z 842.634,A -85,B 0,C 180,E1 24128.538,E2 24128.538} C_VEL
LIN {X 0,Y 200.294,Z 841.728,A -85,B 0,C 180,E1 24137.499,E2 24137.499} C_VEL
LIN {X 0,Y 199.788,Z 843.853,A -85,B 0,C 180,E1 24144.992,E2 24144.992} C_VEL
LIN {X 0,Y 199.422,Z 849.174,A -85,B 0,C 180,E1 24151.935,E2 24151.935} C_VEL
LIN {X 0,Y 198.714,Z 860.08,A -85,B 0,C 180,E1 24160.59,E2 24160.59} C_VEL
LIN {X 0,Y 197.361,Z 870.095,A -85,B 0,C 180,E1 24166.518,E2 24166.518} C_VEL
LIN {X 0,Y 176.448,Z 896.341,A -85,B 0,C 180,E1 24171.682,E2 24171.682} C_VEL
LIN {X 0,Y 152.368,Z 920.603,A -85,B 0,C 180,E1 24179.499,E2 24179.499} C_VEL
LIN {X 0,Y 129.916,Z 939.762,A -85,B 0,C 180,E1 24190.952,E2 24190.952} C_VEL
LIN {X 0,Y 112.56,Z 953.471,A -85,B 0,C 180,E1 24207.442,E2 24207.442} C_VEL
LIN {X 0,Y 104.902,Z 959.876,A -85,B 0,C 180,E1 24222.458,E2 24222.458} C_VEL
LIN {X 0,Y 103.072,Z 963.579,A -85,B 0,C 180,E1 24244.407,E2 24244.407} C_VEL
LIN {X 0,Y 102.54,Z 963.923,A -85,B 0,C 180,E1 24251.679,E2 24251.679} C_VEL
LIN {X 0,Y 102.515,Z 963.552,A -85,B 0,C 180,E1 24262.768,E2 24262.768} C_VEL
LIN {X 0,Y 103.207,Z 963.367,A -85,B 0,C 180,E1 24263.927,E2 24263.927} C_VEL
LIN {X 0,Y 122.352,Z 957.394,A -85,B 0,C 180,E1 24282.252,E2 24282.252} C_VEL
LIN {X 0,Y 148.605,Z 946.152,A -85,B 0,C 180,E1 24294.847,E2 24294.847} C_VEL
LIN {X 0,Y 179.322,Z 929.006,A -85,B 0,C 180,E1 24303.384,E2 24303.384} C_VEL
LIN {X 0,Y 210.031,Z 906.798,A -85,B 0,C 180,E1 24308.917,E2 24308.917} C_VEL
LIN {X 0,Y 217.919,Z 900.125,A -85,B 0,C 180,E1 24310.016,E2 24310.016} C_VEL
LIN {X 0,Y 217.07,Z 901.069,A -85,B 0,C 180,E1 24310.588,E2 24310.588} C_VEL
LIN {X 0,Y 185.803,Z 927.169,A -85,B 0,C 180,E1 24315.322,E2 24315.322} C_VEL
LIN {X 0,Y 153.654,Z 948.671,A -85,B 0,C 180,E1 24322.946,E2 24322.946} C_VEL
LIN {X 0,Y 124.531,Z 964.86,A -85,B 0,C 180,E1 24335.119,E2 24335.119} C_VEL
LIN {X 0,Y 103.141,Z 975.654,A -85,B 0,C 180,E1 24354.179,E2 24354.179} C_VEL
LIN {X 0,Y 95.928,Z 979.786,A -85,B 0,C 180,E1 24371.661,E2 24371.661} C_VEL
LIN {X 0,Y 95.712,Z 980.561,A -85,B 0,C 180,E1 24389.999,E2 24389.999} C_VEL
LIN {X 0,Y 96.541,Z 976.684,A -85,B 0,C 180,E1 24410.135,E2 24410.135} C_VEL
LIN {X 0,Y 107.105,Z 966.81,A -85,B 0,C 180,E1 24430.951,E2 24430.951} C_VEL
LIN {X 0,Y 128.066,Z 950.234,A -85,B 0,C 180,E1 24447.251,E2 24447.251} C_VEL
LIN {X 0,Y 152.975,Z 928.728,A -85,B 0,C 180,E1 24457.636,E2 24457.636} C_VEL
LIN {X 0,Y 177.911,Z 903.032,A -85,B 0,C 180,E1 24464.273,E2 24464.273} C_VEL
LIN {X 0,Y 197.786,Z 877.837,A -85,B 0,C 180,E1 24468.237,E2 24468.237} C_VEL
LIN {X 0,Y 198.452,Z 864.407,A -85,B 0,C 180,E1 24475.605,E2 24475.605} C_VEL
LIN {X 0,Y 198.316,Z 854.103,A -85,B 0,C 180,E1 24483.236,E2 24483.236} C_VEL
LIN {X 0,Y 198.042,Z 849.201,A -85,B 0,C 180,E1 24488.728,E2 24488.728} C_VEL
LIN {X 0,Y 195.883,Z 848.423,A -85,B 0,C 180,E1 24497.906,E2 24497.906} C_VEL
LIN {X 0,Y 195.238,Z 850.826,A -85,B 0,C 180,E1 24505.616,E2 24505.616} C_VEL
LIN {X 0,Y 194.473,Z 856.726,A -85,B 0,C 180,E1 24512.848,E2 24512.848} C_VEL
LIN {X 0,Y 193.346,Z 865.98,A -85,B 0,C 180,E1 24520.251,E2 24520.251} C_VEL
LIN {X 0,Y 191.991,Z 873.565,A -85,B 0,C 180,E1 24524.978,E2 24524.978} C_VEL
LIN {X 0,Y 168.777,Z 900.913,A -85,B 0,C 180,E1 24530.429,E2 24530.429} C_VEL
LIN {X 0,Y 144.228,Z 924.185,A -85,B 0,C 180,E1 24538.458,E2 24538.458} C_VEL
LIN {X 0,Y 120.996,Z 942.572,A -85,B 0,C 180,E1 24550.63,E2 24550.63} C_VEL
LIN {X 0,Y 104.344,Z 954.876,A -85,B 0,C 180,E1 24567.222,E2 24567.222} C_VEL
LIN {X 0,Y 96.578,Z 961.08,A -85,B 0,C 180,E1 24583.556,E2 24583.556} C_VEL
LIN {X 0,Y 95.173,Z 964.213,A -85,B 0,C 180,E1 24604.91,E2 24604.91} C_VEL
LIN {X 0,Y 103.207,Z 963.367,A -85,B 0,C 180,E1 24623.927,E2 24623.927} C_VEL
LIN {X 0,Y 106.112,Z 962.532,A -85,B 0,C 180,E1 24630.928,E2 24630.928} C_VEL
LIN {X 0,Y 111.2,Z 960.402,A -85,B 0,C 180,E1 24641.01,E2 24641.01} C_VEL
LIN {X 0,Y 112.366,Z 959.999,A -85,B 0,C 180,E1 24641.946,E2 24641.946} C_VEL
LIN {X 0,Y 141.138,Z 949.088,A -85,B 0,C 180,E1 24656.291,E2 24656.291} C_VEL
LIN {X 0,Y 173.244,Z 932.625,A -85,B 0,C 180,E1 24665.036,E2 24665.036} C_VEL
LIN {X 0,Y 202.086,Z 913.457,A -85,B 0,C 180,E1 24670.085,E2 24670.085} C_VEL
LIN {X 0,Y 169.36,Z 937.219,A -85,B 0,C 180,E1 24675.543,E2 24675.543} C_VEL
LIN {X 0,Y 136.789,Z 956.173,A -85,B 0,C 180,E1 24684.476,E2 24684.476} C_VEL
LIN {X 0,Y 107.191,Z 970.448,A -85,B 0,C 180,E1 24700.356,E2 24700.356} C_VEL
LIN {X 0,Y 91.462,Z 977.507,A -85,B 0,C 180,E1 24720.331,E2 24720.331} C_VEL
LIN {X 0,Y 87.072,Z 979.868,A -85,B 0,C 180,E1 24740.018,E2 24740.018} C_VEL
LIN {X 0,Y 87.797,Z 979.771,A -85,B 0,C 180,E1 24749.999,E2 24749.999} C_VEL
LIN {X 0,Y 88.574,Z 976.3,A -85,B 0,C 180,E1 24769.92,E2 24769.92} C_VEL
LIN {X 0,Y 98.277,Z 967.69,A -85,B 0,C 180,E1 24790.735,E2 24790.735} C_VEL
LIN {X 0,Y 117.163,Z 953.817,A -85,B 0,C 180,E1 24806.842,E2 24806.842} C_VEL
LIN {X 0,Y 141.913,Z 934.175,A -85,B 0,C 180,E1 24817.978,E2 24817.978} C_VEL
LIN {X 0,Y 168.508,Z 908.937,A -85,B 0,C 180,E1 24825.336,E2 24825.336} C_VEL
LIN {X 0,Y 192.331,Z 880.717,A -85,B 0,C 180,E1 24829.972,E2 24829.972} C_VEL
LIN {X 0,Y 193.298,Z 867.753,A -85,B 0,C 180,E1 24837.728,E2 24837.728} C_VEL
LIN {X 0,Y 193.586,Z 858.35,A -85,B 0,C 180,E1 24845.555,E2 24845.555} C_VEL
LIN {X 0,Y 193.502,Z 855.664,A -85,B 0,C 180,E1 24848.935,E2 24848.935} C_VEL
LIN {X 0,Y 191.26,Z 855.128,A -85,B 0,C 180,E1 24858.777,E2 24858.777} C_VEL
LIN {X 0,Y 190.368,Z 858.074,A -85,B 0,C 180,E1 24866.845,E2 24866.845} C_VEL
LIN {X 0,Y 189.233,Z 864.298,A -85,B 0,C 180,E1 24873.879,E2 24873.879} C_VEL
LIN {X 0,Y 187.359,Z 874.068,A -85,B 0,C 180,E1 24881.461,E2 24881.461} C_VEL
LIN {X 0,Y 186.673,Z 877.012,A -85,B 0,C 180,E1 24883.32,E2 24883.32} C_VEL
LIN {X 0,Y 161.194,Z 905.256,A -85,B 0,C 180,E1 24889.058,E2 24889.058} C_VEL
LIN {X 0,Y 135.913,Z 927.652,A -85,B 0,C 180,E1 24897.363,E2 24897.363} C_VEL
LIN {X 0,Y 114.307,Z 943.702,A -85,B 0,C 180,E1 24908.609,E2 24908.609} C_VEL
LIN {X 0,Y 97.69,Z 955.17,A -85,B 0,C 180,E1 24924.655,E2 24924.655} C_VEL
LIN {X 0,Y 88.273,Z 962.145,A -85,B 0,C 180,E1 24944.664,E2 24944.664} C_VEL
LIN {X 0,Y 86.82,Z 964.718,A -85,B 0,C 180,E1 24961.43,E2 24961.43} C_VEL
LIN {X 0,Y 95.866,Z 964.262,A -85,B 0,C 180,E1 24985.61,E2 24985.61} C_VEL
LIN {X 0,Y 112.366,Z 959.999,A -85,B 0,C 180,E1 25001.946,E2 25001.946} C_VEL
LIN {X 0,Y 120.008,Z 957.196,A -85,B 0,C 180,E1 25009.627,E2 25009.627} C_VEL
LIN {X 0,Y 129.347,Z 953.617,A -85,B 0,C 180,E1 25016.252,E2 25016.252} C_VEL
LIN {X 0,Y 160.822,Z 939.593,A -85,B 0,C 180,E1 25025.426,E2 25025.426} C_VEL
LIN {X 0,Y 183.735,Z 926.59,A -85,B 0,C 180,E1 25029.743,E2 25029.743} C_VEL
LIN {X 0,Y 183.967,Z 926.538,A -85,B 0,C 180,E1 25030.156,E2 25030.156} C_VEL
LIN {X 0,Y 149.675,Z 947.673,A -85,B 0,C 180,E1 25036.703,E2 25036.703} C_VEL
LIN {X 0,Y 118.674,Z 962.939,A -85,B 0,C 180,E1 25047.112,E2 25047.112} C_VEL
LIN {X 0,Y 94.114,Z 973.103,A -85,B 0,C 180,E1 25063.817,E2 25063.817} C_VEL
LIN {X 0,Y 80.752,Z 978.429,A -85,B 0,C 180,E1 25088.052,E2 25088.052} C_VEL
LIN {X 0,Y 79.88,Z 978.977,A -85,B 0,C 180,E1 25109.999,E2 25109.999} C_VEL
LIN {X 0,Y 81.018,Z 975.386,A -85,B 0,C 180,E1 25131.869,E2 25131.869} C_VEL
LIN {X 0,Y 92.197,Z 966.572,A -85,B 0,C 180,E1 25154.075,E2 25154.075} C_VEL
LIN {X 0,Y 112.843,Z 952.453,A -85,B 0,C 180,E1 25170.368,E2 25170.368} C_VEL
LIN {X 0,Y 139.817,Z 931.861,A -85,B 0,C 180,E1 25181.427,E2 25181.427} C_VEL
LIN {X 0,Y 168.052,Z 905.35,A -85,B 0,C 180,E1 25188.382,E2 25188.382} C_VEL
LIN {X 0,Y 186.831,Z 883.391,A -85,B 0,C 180,E1 25191.868,E2 25191.868} C_VEL
LIN {X 0,Y 188.214,Z 871.089,A -85,B 0,C 180,E1 25199.963,E2 25199.963} C_VEL
LIN {X 0,Y 188.702,Z 863.642,A -85,B 0,C 180,E1 25206.851,E2 25206.851} C_VEL
LIN {X 0,Y 188.71,Z 861.947,A -85,B 0,C 180,E1 25209.163,E2 25209.163} C_VEL
LIN {X 0,Y 186.506,Z 861.514,A -85,B 0,C 180,E1 25218.839,E2 25218.839} C_VEL
LIN {X 0,Y 185.536,Z 864.261,A -85,B 0,C 180,E1 25226.536,E2 25226.536} C_VEL
LIN {X 0,Y 183.774,Z 871.581,A -85,B 0,C 180,E1 25234.803,E2 25234.803} C_VEL
LIN {X 0,Y 181.358,Z 880.401,A -85,B 0,C 180,E1 25241.509,E2 25241.509} C_VEL
LIN {X 0,Y 156.847,Z 906.453,A -85,B 0,C 180,E1 25246.726,E2 25246.726} C_VEL
LIN {X 0,Y 130.858,Z 928.567,A -85,B 0,C 180,E1 25254.79,E2 25254.79} C_VEL
LIN {X 0,Y 106.783,Z 945.466,A -85,B 0,C 180,E1 25267.019,E2 25267.019} C_VEL
LIN {X 0,Y 88.702,Z 957.075,A -85,B 0,C 180,E1 25285.308,E2 25285.308} C_VEL
LIN {X 0,Y 81.353,Z 962.04,A -85,B 0,C 180,E1 25300.691,E2 25300.691} C_VEL
LIN {X 0,Y 79.304,Z 965.581,A -85,B 0,C 180,E1 25324.811,E2 25324.811} C_VEL
LIN {X 0,Y 90.607,Z 964.908,A -85,B 0,C 180,E1 25350.12,E2 25350.12} C_VEL
LIN {X 0,Y 115.091,Z 958.63,A -85,B 0,C 180,E1 25369.804,E2 25369.804} C_VEL
LIN {X 0,Y 129.347,Z 953.617,A -85,B 0,C 180,E1 25376.252,E2 25376.252} C_VEL
LIN {X 0,Y 140.013,Z 949.336,A -85,B 0,C 180,E1 25381.894,E2 25381.894} C_VEL
LIN {X 0,Y 149.925,Z 945.133,A -85,B 0,C 180,E1 25386.226,E2 25386.226} C_VEL
LIN {X 0,Y 151.647,Z 944.364,A -85,B 0,C 180,E1 25386.65,E2 25386.65} C_VEL
LIN {X 0,Y 167.294,Z 936.639,A -85,B 0,C 180,E1 25389.76,E2 25389.76} C_VEL
LIN {X 0,Y 130.471,Z 956.053,A -85,B 0,C 180,E1 25398.05,E2 25398.05} C_VEL
LIN {X 0,Y 98.998,Z 968.936,A -85,B 0,C 180,E1 25411.842,E2 25411.842} C_VEL
LIN {X 0,Y 77.705,Z 976.279,A -85,B 0,C 180,E1 25434.365,E2 25434.365} C_VEL
LIN {X 0,Y 71.402,Z 978.365,A -85,B 0,C 180,E1 25457.797,E2 25457.797} C_VEL
LIN {X 0,Y 71.968,Z 978.18,A -85,B 0,C 180,E1 25469.998,E2 25469.998} C_VEL
LIN {X 0,Y 73.573,Z 974.457,A -85,B 0,C 180,E1 25494.216,E2 25494.216} C_VEL
LIN {X 0,Y 88.616,Z 964.146,A -85,B 0,C 180,E1 25520.021,E2 25520.021} C_VEL
LIN {X 0,Y 114.04,Z 947.615,A -85,B 0,C 180,E1 25536.551,E2 25536.551} C_VEL
LIN {X 0,Y 141.891,Z 926.353,A -85,B 0,C 180,E1 25545.901,E2 25545.901} C_VEL
LIN {X 0,Y 169.896,Z 899.684,A -85,B 0,C 180,E1 25551.75,E2 25551.75} C_VEL
LIN {X 0,Y 181.381,Z 886.441,A -85,B 0,C 180,E1 25553.695,E2 25553.695} C_VEL
LIN {X 0,Y 183,Z 875.905,A -85,B 0,C 180,E1 25561.143,E2 25561.143} C_VEL
LIN {X 0,Y 183.705,Z 869.81,A -85,B 0,C 180,E1 25567.038,E2 25567.038} C_VEL
LIN {X 0,Y 183.688,Z 868.14,A -85,B 0,C 180,E1 25569.665,E2 25569.665} C_VEL
LIN {X 0,Y 181.47,Z 867.937,A -85,B 0,C 180,E1 25579.383,E2 25579.383} C_VEL
LIN {X 0,Y 180.232,Z 871.094,A -85,B 0,C 180,E1 25587.381,E2 25587.381} C_VEL
LIN {X 0,Y 177.998,Z 878.393,A -85,B 0,C 180,E1 25595.405,E2 25595.405} C_VEL
LIN {X 0,Y 176.179,Z 883.653,A -85,B 0,C 180,E1 25599.568,E2 25599.568} C_VEL
LIN {X 0,Y 151.117,Z 909.105,A -85,B 0,C 180,E1 25604.645,E2 25604.645} C_VEL
LIN {X 0,Y 124.332,Z 930.742,A -85,B 0,C 180,E1 25612.639,E2 25612.639} C_VEL
LIN {X 0,Y 98.489,Z 947.771,A -85,B 0,C 180,E1 25625.851,E2 25625.851} C_VEL
LIN {X 0,Y 80.541,Z 958.386,A -85,B 0,C 180,E1 25644.626,E2 25644.626} C_VEL
LIN {X 0,Y 72.894,Z 963.226,A -85,B 0,C 180,E1 25661.949,E2 25661.949} C_VEL
LIN {X 0,Y 72.137,Z 966.44,A -85,B 0,C 180,E1 25688.873,E2 25688.873} C_VEL
LIN {X 0,Y 84.385,Z 965.75,A -85,B 0,C 180,E1 25713.4,E2 25713.4} C_VEL
LIN {X 0,Y 108.581,Z 960.307,A -85,B 0,C 180,E1 25732.078,E2 25732.078} C_VEL
LIN {X 0,Y 140.619,Z 949.159,A -85,B 0,C 180,E1 25743.975,E2 25743.975} C_VEL
LIN {X 0,Y 151.647,Z 944.364,A -85,B 0,C 180,E1 25746.65,E2 25746.65} C_VEL
LIN {X 0,Y 151.625,Z 944.566,A -85,B 0,C 180,E1 25748.063,E2 25748.063} C_VEL
LIN {X 0,Y 145.243,Z 947.949,A -85,B 0,C 180,E1 25750.426,E2 25750.426} C_VEL
LIN {X 0,Y 135.502,Z 952.602,A -85,B 0,C 180,E1 25752.755,E2 25752.755} C_VEL
LIN {X 0,Y 99.864,Z 966.843,A -85,B 0,C 180,E1 25764.951,E2 25764.951} C_VEL
LIN {X 0,Y 76.103,Z 974.241,A -85,B 0,C 180,E1 25783.392,E2 25783.392} C_VEL
LIN {X 0,Y 64.243,Z 977.495,A -85,B 0,C 180,E1 25810.26,E2 25810.26} C_VEL
LIN {X 0,Y 64.042,Z 977.378,A -85,B 0,C 180,E1 25829.998,E2 25829.998} C_VEL
LIN {X 0,Y 66.284,Z 973.509,A -85,B 0,C 180,E1 25857.084,E2 25857.084} C_VEL
LIN {X 0,Y 83.565,Z 962.916,A -85,B 0,C 180,E1 25884.35,E2 25884.35} C_VEL
LIN {X 0,Y 110.339,Z 946.529,A -85,B 0,C 180,E1 25900.232,E2 25900.232} C_VEL
LIN {X 0,Y 138.44,Z 925.885,A -85,B 0,C 180,E1 25908.814,E2 25908.814} C_VEL
LIN {X 0,Y 166.835,Z 899.562,A -85,B 0,C 180,E1 25914.233,E2 25914.233} C_VEL
LIN {X 0,Y 176.003,Z 889.428,A -85,B 0,C 180,E1 25915.658,E2 25915.658} C_VEL
LIN {X 0,Y 177.956,Z 879.3,A -85,B 0,C 180,E1 25923.606,E2 25923.606} C_VEL
LIN {X 0,Y 178.669,Z 874.214,A -85,B 0,C 180,E1 25929.683,E2 25929.683} C_VEL
LIN {X 0,Y 176.314,Z 874.243,A -85,B 0,C 180,E1 25939.973,E2 25939.973} C_VEL
LIN {X 0,Y 174.759,Z 877.589,A -85,B 0,C 180,E1 25948.074,E2 25948.074} C_VEL
LIN {X 0,Y 171.899,Z 885.1,A -85,B 0,C 180,E1 25956.037,E2 25956.037} C_VEL
LIN {X 0,Y 171.207,Z 886.888,A -85,B 0,C 180,E1 25957.509,E2 25957.509} C_VEL
LIN {X 0,Y 142.978,Z 913.924,A -85,B 0,C 180,E1 25962.974,E2 25962.974} C_VEL
LIN {X 0,Y 114.818,Z 934.912,A -85,B 0,C 180,E1 25971.384,E2 25971.384} C_VEL
LIN {X 0,Y 89.343,Z 950.331,A -85,B 0,C 180,E1 25985.024,E2 25985.024} C_VEL
LIN {X 0,Y 72.253,Z 959.676,A -85,B 0,C 180,E1 26004.007,E2 26004.007} C_VEL
LIN {X 0,Y 63.526,Z 965.067,A -85,B 0,C 180,E1 26028.551,E2 26028.551} C_VEL
LIN {X 0,Y 66.35,Z 967.393,A -85,B 0,C 180,E1 26057.131,E2 26057.131} C_VEL
LIN {X 0,Y 84.523,Z 965.72,A -85,B 0,C 180,E1 26083.033,E2 26083.033} C_VEL
LIN {X 0,Y 114.8,Z 958.527,A -85,B 0,C 180,E1 26100.06,E2 26100.06} C_VEL
LIN {X 0,Y 148.949,Z 946.023,A -85,B 0,C 180,E1 26109.415,E2 26109.415} C_VEL
LIN {X 0,Y 142.33,Z 949.468,A -85,B 0,C 180,E1 26111.266,E2 26111.266} C_VEL
LIN {X 0,Y 135.502,Z 952.602,A -85,B 0,C 180,E1 26112.755,E2 26112.755} C_VEL
